LIN {X 0,Y 249.229,Z 243.435,A -85,B 0,C 180,E1 -19068.626,E2 -19068.626} C_VEL
LIN {X 0,Y 249.43,Z 243.409,A -85,B 0,C 180,E1 -19071.911,E2 -19071.911} C_VEL
LIN {X 0,Y 249.274,Z 243.427,A -85,B 0,C 180,E1 -19075.157,E2 -19075.157} C_VEL
LIN {X 0,Y 249.658,Z 243.377,A -85,B 0,C 180,E1 -19078.648,E2 -19078.648} C_VEL
LIN {X 0,Y 249.31,Z 243.427,A -85,B 0,C 180,E1 -19079.548,E2 -19079.548} C_VEL
LIN {X 0,Y 247.865,Z 243.609,A -85,B 0,C 180,E1 -19080.873,E2 -19080.873} C_VEL
LIN {X 0,Y 243.339,Z 244.172,A -85,B 0,C 180,E1 -19083.962,E2 -19083.962} C_VEL
LIN {X 0,Y 242.329,Z 244.29,A -85,B 0,C 180,E1 -19085.35,E2 -19085.35} C_VEL
LIN {X 0,Y 242.288,Z 244.292,A -85,B 0,C 180,E1 -19085.821,E2 -19085.821} C_VEL
LIN {X 0,Y 242.33,Z 244.288,A -85,B 0,C 180,E1 -19089.588,E2 -19089.588} C_VEL
LIN {X 0,Y 242.123,Z 244.317,A -85,B 0,C 180,E1 -19095.152,E2 -19095.152} C_VEL
LIN {X 0,Y 242.026,Z 244.326,A -85,B 0,C 180,E1 -19098.637,E2 -19098.637} C_VEL
LIN {X 0,Y 241.979,Z 244.332,A -85,B 0,C 180,E1 -19102.192,E2 -19102.192} C_VEL
LIN {X 0,Y 241.995,Z 244.332,A -85,B 0,C 180,E1 -19105.834,E2 -19105.834} C_VEL
LIN {X 0,Y 241.972,Z 244.336,A -85,B 0,C 180,E1 -19109.597,E2 -19109.597} C_VEL
LIN {X 0,Y 241.979,Z 244.335,A -85,B 0,C 180,E1 -19113.502,E2 -19113.502} C_VEL
LIN {X 0,Y 241.978,Z 244.34,A -85,B 0,C 180,E1 -19117.593,E2 -19117.593} C_VEL
LIN {X 0,Y 241.892,Z 244.354,A -85,B 0,C 180,E1 -19121.942,E2 -19121.942} C_VEL
LIN {X 0,Y 241.926,Z 244.377,A -85,B 0,C 180,E1 -19125.083,E2 -19125.083} C_VEL
LIN {X 0,Y 244.497,Z 252.638,A -85,B 0,C 180,E1 -19129.628,E2 -19129.628} C_VEL
LIN {X 0,Y 245.734,Z 256.877,A -85,B 0,C 180,E1 -19131.703,E2 -19131.703} C_VEL
LIN {X 0,Y 248.18,Z 261.171,A -85,B 0,C 180,E1 -19132.469,E2 -19132.469} C_VEL
LIN {X 0,Y 251.912,Z 267.851,A -85,B 0,C 180,E1 -19133.592,E2 -19133.592} C_VEL
LIN {X 0,Y 258.214,Z 280.37,A -85,B 0,C 180,E1 -19135.402,E2 -19135.402} C_VEL
LIN {X 0,Y 262.949,Z 291.618,A -85,B 0,C 180,E1 -19136.722,E2 -19136.722} C_VEL
LIN {X 0,Y 265.386,Z 308.755,A -85,B 0,C 180,E1 -19137.801,E2 -19137.801} C_VEL
LIN {X 0,Y 265.835,Z 312.992,A -85,B 0,C 180,E1 -19138.034,E2 -19138.034} C_VEL
LIN {X 0,Y 263.208,Z 366.769,A -85,B 0,C 180,E1 -19139.626,E2 -19139.626} C_VEL
LIN {X 0,Y 261.857,Z 380.21,A -85,B 0,C 180,E1 -19140.286,E2 -19140.286} C_VEL
LIN {X 0,Y 260.056,Z 392.016,A -85,B 0,C 180,E1 -19141.115,E2 -19141.115} C_VEL
LIN {X 0,Y 257.961,Z 403.306,A -85,B 0,C 180,E1 -19142.19,E2 -19142.19} C_VEL
LIN {X 0,Y 255.717,Z 413.719,A -85,B 0,C 180,E1 -19143.475,E2 -19143.475} C_VEL
LIN {X 0,Y 252.935,Z 424.487,A -85,B 0,C 180,E1 -19145.15,E2 -19145.15} C_VEL
LIN {X 0,Y 250.015,Z 435.103,A -85,B 0,C 180,E1 -19147.263,E2 -19147.263} C_VEL
LIN {X 0,Y 247.678,Z 442.971,A -85,B 0,C 180,E1 -19149.227,E2 -19149.227} C_VEL
LIN {X 0,Y 245.365,Z 450.7,A -85,B 0,C 180,E1 -19151.635,E2 -19151.635} C_VEL
LIN {X 0,Y 243.433,Z 456.957,A -85,B 0,C 180,E1 -19154.082,E2 -19154.082} C_VEL
LIN {X 0,Y 241.818,Z 461.955,A -85,B 0,C 180,E1 -19156.556,E2 -19156.556} C_VEL
LIN {X 0,Y 240.833,Z 465.839,A -85,B 0,C 180,E1 -19159.066,E2 -19159.066} C_VEL
LIN {X 0,Y 240.18,Z 468.71,A -85,B 0,C 180,E1 -19161.587,E2 -19161.587} C_VEL
LIN {X 0,Y 239.825,Z 471.07,A -85,B 0,C 180,E1 -19164.957,E2 -19164.957} C_VEL
LIN {X 0,Y 239.808,Z 471.654,A -85,B 0,C 180,E1 -19166.64,E2 -19166.64} C_VEL
LIN {X 0,Y 239.888,Z 471.802,A -85,B 0,C 180,E1 -19168.321,E2 -19168.321} C_VEL
LIN {X 0,Y 239.955,Z 471.553,A -85,B 0,C 180,E1 -19170,E2 -19170} C_VEL
LIN {X 0,Y 239.918,Z 470.902,A -85,B 0,C 180,E1 -19171.679,E2 -19171.679} C_VEL
LIN {X 0,Y 239.837,Z 469.834,A -85,B 0,C 180,E1 -19173.36,E2 -19173.36} C_VEL
LIN {X 0,Y 239.866,Z 468.298,A -85,B 0,C 180,E1 -19175.043,E2 -19175.043} C_VEL
LIN {X 0,Y 240.061,Z 465.178,A -85,B 0,C 180,E1 -19177.57,E2 -19177.57} C_VEL
LIN {X 0,Y 240.512,Z 460.957,A -85,B 0,C 180,E1 -19180.097,E2 -19180.097} C_VEL
LIN {X 0,Y 241.43,Z 454.492,A -85,B 0,C 180,E1 -19183.038,E2 -19183.038} C_VEL
LIN {X 0,Y 242.788,Z 447.431,A -85,B 0,C 180,E1 -19185.531,E2 -19185.531} C_VEL
LIN {X 0,Y 244.421,Z 438.541,A -85,B 0,C 180,E1 -19188.005,E2 -19188.005} C_VEL
LIN {X 0,Y 246.24,Z 428.427,A -85,B 0,C 180,E1 -19190.246,E2 -19190.246} C_VEL
LIN {X 0,Y 248.041,Z 418.09,A -85,B 0,C 180,E1 -19192.05,E2 -19192.05} C_VEL
LIN {X 0,Y 249.916,Z 406.654,A -85,B 0,C 180,E1 -19193.623,E2 -19193.623} C_VEL
LIN {X 0,Y 251.607,Z 394.804,A -85,B 0,C 180,E1 -19194.88,E2 -19194.88} C_VEL
LIN {X 0,Y 252.985,Z 382.547,A -85,B 0,C 180,E1 -19195.836,E2 -19195.836} C_VEL
LIN {X 0,Y 254.124,Z 368.734,A -85,B 0,C 180,E1 -19196.563,E2 -19196.563} C_VEL
LIN {X 0,Y 256.185,Z 310.245,A -85,B 0,C 180,E1 -19198.329,E2 -19198.329} C_VEL
LIN {X 0,Y 251.646,Z 276.723,A -85,B 0,C 180,E1 -19199.901,E2 -19199.901} C_VEL
LIN {X 0,Y 245.317,Z 259.472,A -85,B 0,C 180,E1 -19201.221,E2 -19201.221} C_VEL
LIN {X 0,Y 243.089,Z 248.916,A -85,B 0,C 180,E1 -19205.325,E2 -19205.325} C_VEL
LIN {X 0,Y 242.019,Z 244.338,A -85,B 0,C 180,E1 -19207.219,E2 -19207.219} C_VEL
LIN {X 0,Y 241.893,Z 244.353,A -85,B 0,C 180,E1 -19211.931,E2 -19211.931} C_VEL
LIN {X 0,Y 241.896,Z 244.354,A -85,B 0,C 180,E1 -19216.579,E2 -19216.579} C_VEL
LIN {X 0,Y 241.988,Z 244.344,A -85,B 0,C 180,E1 -19221.641,E2 -19221.641} C_VEL
LIN {X 0,Y 241.987,Z 244.341,A -85,B 0,C 180,E1 -19224.48,E2 -19224.48} C_VEL
LIN {X 0,Y 241.94,Z 244.345,A -85,B 0,C 180,E1 -19228.466,E2 -19228.466} C_VEL
LIN {X 0,Y 241.96,Z 244.343,A -85,B 0,C 180,E1 -19232.298,E2 -19232.298} C_VEL
LIN {X 0,Y 241.989,Z 244.342,A -85,B 0,C 180,E1 -19236,E2 -19236} C_VEL
LIN {X 0,Y 241.989,Z 244.332,A -85,B 0,C 180,E1 -19239.595,E2 -19239.595} C_VEL
LIN {X 0,Y 242.118,Z 244.307,A -85,B 0,C 180,E1 -19243.31,E2 -19243.31} C_VEL
LIN {X 0,Y 242.161,Z 244.319,A -85,B 0,C 180,E1 -19248.27,E2 -19248.27} C_VEL
LIN {X 0,Y 242.356,Z 244.29,A -85,B 0,C 180,E1 -19251.654,E2 -19251.654} C_VEL
LIN {X 0,Y 242.386,Z 244.28,A -85,B 0,C 180,E1 -19253.331,E2 -19253.331} C_VEL
LIN {X 0,Y 242.601,Z 244.245,A -85,B 0,C 180,E1 -19258.331,E2 -19258.331} C_VEL
LIN {X 0,Y 242.609,Z 244.26,A -85,B 0,C 180,E1 -19261.651,E2 -19261.651} C_VEL
LIN {X 0,Y 242.383,Z 244.29,A -85,B 0,C 180,E1 -19266.65,E2 -19266.65} C_VEL
LIN {X 0,Y 242.253,Z 244.302,A -85,B 0,C 180,E1 -19270.014,E2 -19270.014} C_VEL
LIN {X 0,Y 242.121,Z 244.325,A -85,B 0,C 180,E1 -19275.133,E2 -19275.133} C_VEL
LIN {X 0,Y 242.04,Z 244.325,A -85,B 0,C 180,E1 -19278.616,E2 -19278.616} C_VEL
LIN {X 0,Y 241.984,Z 244.339,A -85,B 0,C 180,E1 -19282.171,E2 -19282.171} C_VEL
LIN {X 0,Y 242.025,Z 244.331,A -85,B 0,C 180,E1 -19285.82,E2 -19285.82} C_VEL
LIN {X 0,Y 241.947,Z 244.323,A -85,B 0,C 180,E1 -19289.579,E2 -19289.579} C_VEL
LIN {X 0,Y 241.948,Z 244.325,A -85,B 0,C 180,E1 -19293.484,E2 -19293.484} C_VEL
LIN {X 0,Y 241.95,Z 244.346,A -85,B 0,C 180,E1 -19297.574,E2 -19297.574} C_VEL
LIN {X 0,Y 241.897,Z 244.349,A -85,B 0,C 180,E1 -19301.915,E2 -19301.915} C_VEL
LIN {X 0,Y 241.896,Z 244.352,A -85,B 0,C 180,E1 -19306.563,E2 -19306.563} C_VEL
LIN {X 0,Y 241.914,Z 244.344,A -85,B 0,C 180,E1 -19310.274,E2 -19310.274} C_VEL
LIN {X 0,Y 241.942,Z 244.347,A -85,B 0,C 180,E1 -19314.483,E2 -19314.483} C_VEL
LIN {X 0,Y 241.928,Z 244.349,A -85,B 0,C 180,E1 -19318.474,E2 -19318.474} C_VEL
LIN {X 0,Y 241.962,Z 244.342,A -85,B 0,C 180,E1 -19322.308,E2 -19322.308} C_VEL
LIN {X 0,Y 242.03,Z 244.338,A -85,B 0,C 180,E1 -19326.014,E2 -19326.014} C_VEL
LIN {X 0,Y 242.033,Z 244.34,A -85,B 0,C 180,E1 -19329.608,E2 -19329.608} C_VEL
LIN {X 0,Y 242.112,Z 244.33,A -85,B 0,C 180,E1 -19333.275,E2 -19333.275} C_VEL
LIN {X 0,Y 242.132,Z 244.324,A -85,B 0,C 180,E1 -19338.277,E2 -19338.277} C_VEL
LIN {X 0,Y 242.374,Z 244.292,A -85,B 0,C 180,E1 -19341.664,E2 -19341.664} C_VEL
LIN {X 0,Y 242.215,Z 244.316,A -85,B 0,C 180,E1 -19345.006,E2 -19345.006} C_VEL
LIN {X 0,Y 242.591,Z 244.267,A -85,B 0,C 180,E1 -19348.34,E2 -19348.34} C_VEL
LIN {X 0,Y 242.586,Z 244.266,A -85,B 0,C 180,E1 -19351.608,E2 -19351.608} C_VEL
LIN {X 0,Y 243.555,Z 247.129,A -85,B 0,C 180,E1 -19351.832,E2 -19351.832} C_VEL
LIN {X 0,Y 252.279,Z 267.97,A -85,B 0,C 180,E1 -19353.517,E2 -19353.517} C_VEL
LIN {X 0,Y 257.026,Z 281.714,A -85,B 0,C 180,E1 -19354.454,E2 -19354.454} C_VEL
LIN {X 0,Y 254.486,Z 350.902,A -85,B 0,C 180,E1 -19356.523,E2 -19356.523} C_VEL
LIN {X 0,Y 253.477,Z 364.221,A -85,B 0,C 180,E1 -19357.225,E2 -19357.225} C_VEL
LIN {X 0,Y 252.336,Z 376.71,A -85,B 0,C 180,E1 -19358.206,E2 -19358.206} C_VEL
LIN {X 0,Y 250.849,Z 388.621,A -85,B 0,C 180,E1 -19359.474,E2 -19359.474} C_VEL
LIN {X 0,Y 249.113,Z 400.327,A -85,B 0,C 180,E1 -19361.088,E2 -19361.088} C_VEL
LIN {X 0,Y 247.294,Z 410.881,A -85,B 0,C 180,E1 -19362.932,E2 -19362.932} C_VEL
LIN {X 0,Y 245.507,Z 420.027,A -85,B 0,C 180,E1 -19364.929,E2 -19364.929} C_VEL
LIN {X 0,Y 243.923,Z 428.643,A -85,B 0,C 180,E1 -19367.275,E2 -19367.275} C_VEL
LIN {X 0,Y 242.477,Z 436.333,A -85,B 0,C 180,E1 -19369.911,E2 -19369.911} C_VEL
LIN {X 0,Y 241.496,Z 441.691,A -85,B 0,C 180,E1 -19372.229,E2 -19372.229} C_VEL
LIN {X 0,Y 240.637,Z 446.89,A -85,B 0,C 180,E1 -19375.155,E2 -19375.155} C_VEL
LIN {X 0,Y 240.121,Z 450.46,A -85,B 0,C 180,E1 -19377.923,E2 -19377.923} C_VEL
LIN {X 0,Y 239.71,Z 452.285,A -85,B 0,C 180,E1 -19379.895,E2 -19379.895} C_VEL
LIN {X 0,Y 239.579,Z 453.5,A -85,B 0,C 180,E1 -19381.871,E2 -19381.871} C_VEL
LIN {X 0,Y 239.59,Z 454.308,A -85,B 0,C 180,E1 -19384.803,E2 -19384.803} C_VEL
LIN {X 0,Y 240.039,Z 453.824,A -85,B 0,C 180,E1 -19387.94,E2 -19387.94} C_VEL
LIN {X 0,Y 240.734,Z 452.276,A -85,B 0,C 180,E1 -19390.638,E2 -19390.638} C_VEL
LIN {X 0,Y 241.725,Z 449.574,A -85,B 0,C 180,E1 -19393.394,E2 -19393.394} C_VEL
LIN {X 0,Y 243.197,Z 445.448,A -85,B 0,C 180,E1 -19396.256,E2 -19396.256} C_VEL
LIN {X 0,Y 244.833,Z 440.722,A -85,B 0,C 180,E1 -19398.699,E2 -19398.699} C_VEL
LIN {X 0,Y 246.897,Z 434.429,A -85,B 0,C 180,E1 -19401.242,E2 -19401.242} C_VEL
LIN {X 0,Y 249.516,Z 426.429,A -85,B 0,C 180,E1 -19403.75,E2 -19403.75} C_VEL
LIN {X 0,Y 252.011,Z 418.028,A -85,B 0,C 180,E1 -19405.837,E2 -19405.837} C_VEL
LIN {X 0,Y 254.554,Z 408.571,A -85,B 0,C 180,E1 -19407.726,E2 -19407.726} C_VEL
LIN {X 0,Y 256.971,Z 398.534,A -85,B 0,C 180,E1 -19409.329,E2 -19409.329} C_VEL
LIN {X 0,Y 259.354,Z 386.633,A -85,B 0,C 180,E1 -19410.818,E2 -19410.818} C_VEL
LIN {X 0,Y 261.389,Z 374.238,A -85,B 0,C 180,E1 -19411.988,E2 -19411.988} C_VEL
LIN {X 0,Y 262.934,Z 361.377,A -85,B 0,C 180,E1 -19412.868,E2 -19412.868} C_VEL
LIN {X 0,Y 264.034,Z 347.279,A -85,B 0,C 180,E1 -19413.476,E2 -19413.476} C_VEL
LIN {X 0,Y 266.847,Z 289.944,A -85,B 0,C 180,E1 -19415.15,E2 -19415.15} C_VEL
LIN {X 0,Y 261.533,Z 277.793,A -85,B 0,C 180,E1 -19416.568,E2 -19416.568} C_VEL
LIN {X 0,Y 255.253,Z 265.81,A -85,B 0,C 180,E1 -19418.282,E2 -19418.282} C_VEL
LIN {X 0,Y 248.063,Z 253.948,A -85,B 0,C 180,E1 -19420.373,E2 -19420.373} C_VEL
LIN {X 0,Y 244.555,Z 248.894,A -85,B 0,C 180,E1 -19421.452,E2 -19421.452} C_VEL
LIN {X 0,Y 242.697,Z 246.476,A -85,B 0,C 180,E1 -19422.037,E2 -19422.037} C_VEL
LIN {X 0,Y 242.208,Z 245.036,A -85,B 0,C 180,E1 -19422.273,E2 -19422.273} C_VEL
LIN {X 0,Y 242.093,Z 244.327,A -85,B 0,C 180,E1 -19422.7,E2 -19422.7} C_VEL
LIN {X 0,Y 242.148,Z 244.324,A -85,B 0,C 180,E1 -19426.585,E2 -19426.585} C_VEL
LIN {X 0,Y 242.378,Z 244.286,A -85,B 0,C 180,E1 -19431.674,E2 -19431.674} C_VEL
LIN {X 0,Y 242.234,Z 244.304,A -85,B 0,C 180,E1 -19435.016,E2 -19435.016} C_VEL
LIN {X 0,Y 242.618,Z 244.254,A -85,B 0,C 180,E1 -19438.643,E2 -19438.643} C_VEL
LIN {X 0,Y 242.615,Z 244.254,A -85,B 0,C 180,E1 -19441.669,E2 -19441.669} C_VEL
LIN {X 0,Y 242.288,Z 244.292,A -85,B 0,C 180,E1 -19445.821,E2 -19445.821} C_VEL
LIN {X 0,Y 241.702,Z 244.374,A -85,B 0,C 180,E1 -19447.208,E2 -19447.208} C_VEL
LIN {X 0,Y 240.104,Z 244.573,A -85,B 0,C 180,E1 -19448.569,E2 -19448.569} C_VEL
LIN {X 0,Y 236.234,Z 245.053,A -85,B 0,C 180,E1 -19451.309,E2 -19451.309} C_VEL
LIN {X 0,Y 235.142,Z 245.192,A -85,B 0,C 180,E1 -19452.743,E2 -19452.743} C_VEL
LIN {X 0,Y 235.058,Z 245.195,A -85,B 0,C 180,E1 -19453.229,E2 -19453.229} C_VEL
LIN {X 0,Y 235.012,Z 245.205,A -85,B 0,C 180,E1 -19457.41,E2 -19457.41} C_VEL
LIN {X 0,Y 234.964,Z 245.207,A -85,B 0,C 180,E1 -19461.996,E2 -19461.996} C_VEL
LIN {X 0,Y 234.914,Z 245.212,A -85,B 0,C 180,E1 -19466.673,E2 -19466.673} C_VEL
LIN {X 0,Y 234.897,Z 245.216,A -85,B 0,C 180,E1 -19470.582,E2 -19470.582} C_VEL
LIN {X 0,Y 234.91,Z 245.22,A -85,B 0,C 180,E1 -19474.651,E2 -19474.651} C_VEL
LIN {X 0,Y 234.927,Z 245.22,A -85,B 0,C 180,E1 -19478.942,E2 -19478.942} C_VEL
LIN {X 0,Y 234.87,Z 245.246,A -85,B 0,C 180,E1 -19483.368,E2 -19483.368} C_VEL
LIN {X 0,Y 237.181,Z 252.68,A -85,B 0,C 180,E1 -19487.809,E2 -19487.809} C_VEL
LIN {X 0,Y 238.401,Z 256.511,A -85,B 0,C 180,E1 -19489.819,E2 -19489.819} C_VEL
LIN {X 0,Y 241.18,Z 261.188,A -85,B 0,C 180,E1 -19490.774,E2 -19490.774} C_VEL
LIN {X 0,Y 245.485,Z 268.562,A -85,B 0,C 180,E1 -19492.18,E2 -19492.18} C_VEL
LIN {X 0,Y 251.778,Z 280.727,A -85,B 0,C 180,E1 -19494.115,E2 -19494.115} C_VEL
LIN {X 0,Y 256.961,Z 292.597,A -85,B 0,C 180,E1 -19495.651,E2 -19495.651} C_VEL
LIN {X 0,Y 257.774,Z 294.794,A -85,B 0,C 180,E1 -19495.893,E2 -19495.893} C_VEL
LIN {X 0,Y 260.076,Z 312.12,A -85,B 0,C 180,E1 -19496.998,E2 -19496.998} C_VEL
LIN {X 0,Y 260.14,Z 316.366,A -85,B 0,C 180,E1 -19497.174,E2 -19497.174} C_VEL
LIN {X 0,Y 257.469,Z 367.039,A -85,B 0,C 180,E1 -19498.714,E2 -19498.714} C_VEL
LIN {X 0,Y 255.975,Z 380.852,A -85,B 0,C 180,E1 -19499.418,E2 -19499.418} C_VEL
LIN {X 0,Y 253.918,Z 393.449,A -85,B 0,C 180,E1 -19500.348,E2 -19500.348} C_VEL
LIN {X 0,Y 251.393,Z 405.87,A -85,B 0,C 180,E1 -19501.625,E2 -19501.625} C_VEL
LIN {X 0,Y 248.783,Z 417.027,A -85,B 0,C 180,E1 -19503.129,E2 -19503.129} C_VEL
LIN {X 0,Y 245.965,Z 427.167,A -85,B 0,C 180,E1 -19504.849,E2 -19504.849} C_VEL
LIN {X 0,Y 242.973,Z 437.148,A -85,B 0,C 180,E1 -19507.016,E2 -19507.016} C_VEL
LIN {X 0,Y 240.25,Z 445.98,A -85,B 0,C 180,E1 -19509.45,E2 -19509.45} C_VEL
LIN {X 0,Y 237.974,Z 453.091,A -85,B 0,C 180,E1 -19511.936,E2 -19511.936} C_VEL
LIN {X 0,Y 235.983,Z 458.809,A -85,B 0,C 180,E1 -19514.453,E2 -19514.453} C_VEL
LIN {X 0,Y 234.503,Z 463.345,A -85,B 0,C 180,E1 -19517.011,E2 -19517.011} C_VEL
LIN {X 0,Y 233.574,Z 466.825,A -85,B 0,C 180,E1 -19519.6,E2 -19519.6} C_VEL
LIN {X 0,Y 232.843,Z 469.921,A -85,B 0,C 180,E1 -19523.066,E2 -19523.066} C_VEL
LIN {X 0,Y 232.714,Z 471.074,A -85,B 0,C 180,E1 -19525.356,E2 -19525.356} C_VEL
LIN {X 0,Y 232.798,Z 471.522,A -85,B 0,C 180,E1 -19528.27,E2 -19528.27} C_VEL
LIN {X 0,Y 232.886,Z 471.246,A -85,B 0,C 180,E1 -19530,E2 -19530} C_VEL
LIN {X 0,Y 232.827,Z 470.566,A -85,B 0,C 180,E1 -19531.73,E2 -19531.73} C_VEL
LIN {X 0,Y 232.784,Z 468.23,A -85,B 0,C 180,E1 -19534.853,E2 -19534.853} C_VEL
LIN {X 0,Y 233.013,Z 464.69,A -85,B 0,C 180,E1 -19537.801,E2 -19537.801} C_VEL
LIN {X 0,Y 233.49,Z 460.401,A -85,B 0,C 180,E1 -19540.404,E2 -19540.404} C_VEL
LIN {X 0,Y 234.463,Z 453.861,A -85,B 0,C 180,E1 -19543.433,E2 -19543.433} C_VEL
LIN {X 0,Y 235.873,Z 446.672,A -85,B 0,C 180,E1 -19545.998,E2 -19545.998} C_VEL
LIN {X 0,Y 237.483,Z 438.386,A -85,B 0,C 180,E1 -19548.358,E2 -19548.358} C_VEL
LIN {X 0,Y 239.355,Z 428.438,A -85,B 0,C 180,E1 -19550.63,E2 -19550.63} C_VEL
LIN {X 0,Y 241.193,Z 418.173,A -85,B 0,C 180,E1 -19552.485,E2 -19552.485} C_VEL
LIN {X 0,Y 243.132,Z 406.814,A -85,B 0,C 180,E1 -19554.097,E2 -19554.097} C_VEL
LIN {X 0,Y 244.87,Z 395.08,A -85,B 0,C 180,E1 -19555.386,E2 -19555.386} C_VEL
LIN {X 0,Y 246.366,Z 382.338,A -85,B 0,C 180,E1 -19556.412,E2 -19556.412} C_VEL
LIN {X 0,Y 247.517,Z 368.578,A -85,B 0,C 180,E1 -19557.158,E2 -19557.158} C_VEL
LIN {X 0,Y 249.654,Z 310.988,A -85,B 0,C 180,E1 -19558.942,E2 -19558.942} C_VEL
LIN {X 0,Y 245.413,Z 278.997,A -85,B 0,C 180,E1 -19560.483,E2 -19560.483} C_VEL
LIN {X 0,Y 238,Z 259.227,A -85,B 0,C 180,E1 -19562.068,E2 -19562.068} C_VEL
LIN {X 0,Y 235.926,Z 249.303,A -85,B 0,C 180,E1 -19566.067,E2 -19566.067} C_VEL
LIN {X 0,Y 234.962,Z 245.217,A -85,B 0,C 180,E1 -19567.819,E2 -19567.819} C_VEL
LIN {X 0,Y 234.843,Z 245.232,A -85,B 0,C 180,E1 -19571.558,E2 -19571.558} C_VEL
LIN {X 0,Y 234.861,Z 245.233,A -85,B 0,C 180,E1 -19575.903,E2 -19575.903} C_VEL
LIN {X 0,Y 234.934,Z 245.22,A -85,B 0,C 180,E1 -19581.072,E2 -19581.072} C_VEL
LIN {X 0,Y 234.911,Z 245.224,A -85,B 0,C 180,E1 -19585.349,E2 -19585.349} C_VEL
LIN {X 0,Y 234.897,Z 245.225,A -85,B 0,C 180,E1 -19589.418,E2 -19589.418} C_VEL
LIN {X 0,Y 234.949,Z 245.217,A -85,B 0,C 180,E1 -19593.814,E2 -19593.814} C_VEL
LIN {X 0,Y 234.942,Z 245.214,A -85,B 0,C 180,E1 -19598.954,E2 -19598.954} C_VEL
LIN {X 0,Y 235.06,Z 245.184,A -85,B 0,C 180,E1 -19603.085,E2 -19603.085} C_VEL
LIN {X 0,Y 235.094,Z 245.201,A -85,B 0,C 180,E1 -19607.912,E2 -19607.912} C_VEL
LIN {X 0,Y 235.295,Z 245.172,A -85,B 0,C 180,E1 -19611.402,E2 -19611.402} C_VEL
LIN {X 0,Y 235.337,Z 245.159,A -85,B 0,C 180,E1 -19613.13,E2 -19613.13} C_VEL
LIN {X 0,Y 235.559,Z 245.121,A -85,B 0,C 180,E1 -19618.281,E2 -19618.281} C_VEL
LIN {X 0,Y 235.568,Z 245.136,A -85,B 0,C 180,E1 -19621.7,E2 -19621.7} C_VEL
LIN {X 0,Y 235.335,Z 245.168,A -85,B 0,C 180,E1 -19626.851,E2 -19626.851} C_VEL
LIN {X 0,Y 235.199,Z 245.18,A -85,B 0,C 180,E1 -19630.318,E2 -19630.318} C_VEL
LIN {X 0,Y 235.068,Z 245.202,A -85,B 0,C 180,E1 -19635.598,E2 -19635.598} C_VEL
LIN {X 0,Y 234.979,Z 245.206,A -85,B 0,C 180,E1 -19639.197,E2 -19639.197} C_VEL
LIN {X 0,Y 234.929,Z 245.219,A -85,B 0,C 180,E1 -19642.874,E2 -19642.874} C_VEL
LIN {X 0,Y 234.931,Z 245.213,A -85,B 0,C 180,E1 -19646.65,E2 -19646.65} C_VEL
LIN {X 0,Y 234.873,Z 245.199,A -85,B 0,C 180,E1 -19650.563,E2 -19650.563} C_VEL
LIN {X 0,Y 234.894,Z 245.209,A -85,B 0,C 180,E1 -19654.63,E2 -19654.63} C_VEL
LIN {X 0,Y 234.878,Z 245.226,A -85,B 0,C 180,E1 -19658.927,E2 -19658.927} C_VEL
LIN {X 0,Y 234.85,Z 245.226,A -85,B 0,C 180,E1 -19663.478,E2 -19663.478} C_VEL
LIN {X 0,Y 234.849,Z 245.229,A -85,B 0,C 180,E1 -19666.507,E2 -19666.507} C_VEL
LIN {X 0,Y 234.876,Z 245.223,A -85,B 0,C 180,E1 -19671.071,E2 -19671.071} C_VEL
LIN {X 0,Y 234.885,Z 245.226,A -85,B 0,C 180,E1 -19675.355,E2 -19675.355} C_VEL
LIN {X 0,Y 234.885,Z 245.23,A -85,B 0,C 180,E1 -19679.426,E2 -19679.426} C_VEL
LIN {X 0,Y 234.947,Z 245.221,A -85,B 0,C 180,E1 -19683.789,E2 -19683.789} C_VEL
LIN {X 0,Y 234.999,Z 245.215,A -85,B 0,C 180,E1 -19688.969,E2 -19688.969} C_VEL
LIN {X 0,Y 235.066,Z 245.205,A -85,B 0,C 180,E1 -19693.04,E2 -19693.04} C_VEL
LIN {X 0,Y 235.064,Z 245.204,A -85,B 0,C 180,E1 -19697.92,E2 -19697.92} C_VEL
LIN {X 0,Y 235.324,Z 245.172,A -85,B 0,C 180,E1 -19701.412,E2 -19701.412} C_VEL
LIN {X 0,Y 235.351,Z 245.165,A -85,B 0,C 180,E1 -19703.14,E2 -19703.14} C_VEL
LIN {X 0,Y 235.551,Z 245.144,A -85,B 0,C 180,E1 -19708.29,E2 -19708.29} C_VEL
LIN {X 0,Y 235.566,Z 245.143,A -85,B 0,C 180,E1 -19710.801,E2 -19710.801} C_VEL
LIN {X 0,Y 236.659,Z 248.134,A -85,B 0,C 180,E1 -19711.049,E2 -19711.049} C_VEL
LIN {X 0,Y 244.391,Z 266.1,A -85,B 0,C 180,E1 -19712.599,E2 -19712.599} C_VEL
LIN {X 0,Y 250.582,Z 283.441,A -85,B 0,C 180,E1 -19713.863,E2 -19713.863} C_VEL
LIN {X 0,Y 247.871,Z 351.487,A -85,B 0,C 180,E1 -19715.945,E2 -19715.945} C_VEL
LIN {X 0,Y 246.857,Z 364.37,A -85,B 0,C 180,E1 -19716.641,E2 -19716.641} C_VEL
LIN {X 0,Y 245.626,Z 377.501,A -85,B 0,C 180,E1 -19717.707,E2 -19717.707} C_VEL
LIN {X 0,Y 243.955,Z 390.157,A -85,B 0,C 180,E1 -19719.116,E2 -19719.116} C_VEL
LIN {X 0,Y 242.261,Z 401.018,A -85,B 0,C 180,E1 -19720.677,E2 -19720.677} C_VEL
LIN {X 0,Y 240.488,Z 410.874,A -85,B 0,C 180,E1 -19722.446,E2 -19722.446} C_VEL
LIN {X 0,Y 238.529,Z 420.706,A -85,B 0,C 180,E1 -19724.66,E2 -19724.66} C_VEL
LIN {X 0,Y 236.756,Z 429.889,A -85,B 0,C 180,E1 -19727.268,E2 -19727.268} C_VEL
LIN {X 0,Y 235.486,Z 436.457,A -85,B 0,C 180,E1 -19729.618,E2 -19729.618} C_VEL
LIN {X 0,Y 234.348,Z 442.397,A -85,B 0,C 180,E1 -19732.293,E2 -19732.293} C_VEL
LIN {X 0,Y 233.481,Z 447.737,A -85,B 0,C 180,E1 -19735.471,E2 -19735.471} C_VEL
LIN {X 0,Y 233.029,Z 450.666,A -85,B 0,C 180,E1 -19737.869,E2 -19737.869} C_VEL
LIN {X 0,Y 232.516,Z 453.203,A -85,B 0,C 180,E1 -19740.919,E2 -19740.919} C_VEL
LIN {X 0,Y 232.459,Z 454.16,A -85,B 0,C 180,E1 -19742.969,E2 -19742.969} C_VEL
LIN {X 0,Y 232.541,Z 454.605,A -85,B 0,C 180,E1 -19745.334,E2 -19745.334} C_VEL
LIN {X 0,Y 233.025,Z 454.036,A -85,B 0,C 180,E1 -19748.377,E2 -19748.377} C_VEL
LIN {X 0,Y 233.864,Z 452.253,A -85,B 0,C 180,E1 -19751.385,E2 -19751.385} C_VEL
LIN {X 0,Y 234.986,Z 449.497,A -85,B 0,C 180,E1 -19754.145,E2 -19754.145} C_VEL
LIN {X 0,Y 236.431,Z 445.601,A -85,B 0,C 180,E1 -19756.884,E2 -19756.884} C_VEL
LIN {X 0,Y 238.36,Z 440.461,A -85,B 0,C 180,E1 -19759.574,E2 -19759.574} C_VEL
LIN {X 0,Y 240.633,Z 434.014,A -85,B 0,C 180,E1 -19762.184,E2 -19762.184} C_VEL
LIN {X 0,Y 243.428,Z 425.799,A -85,B 0,C 180,E1 -19764.745,E2 -19764.745} C_VEL
LIN {X 0,Y 246.242,Z 416.682,A -85,B 0,C 180,E1 -19766.992,E2 -19766.992} C_VEL
LIN {X 0,Y 249.052,Z 406.603,A -85,B 0,C 180,E1 -19768.948,E2 -19768.948} C_VEL
LIN {X 0,Y 251.411,Z 396.809,A -85,B 0,C 180,E1 -19770.465,E2 -19770.465} C_VEL
LIN {X 0,Y 253.85,Z 384.799,A -85,B 0,C 180,E1 -19771.935,E2 -19771.935} C_VEL
LIN {X 0,Y 255.814,Z 373.071,A -85,B 0,C 180,E1 -19773.016,E2 -19773.016} C_VEL
LIN {X 0,Y 257.416,Z 359.361,A -85,B 0,C 180,E1 -19773.919,E2 -19773.919} C_VEL
LIN {X 0,Y 258.443,Z 346.379,A -85,B 0,C 180,E1 -19774.453,E2 -19774.453} C_VEL
LIN {X 0,Y 261.287,Z 292.209,A -85,B 0,C 180,E1 -19776.05,E2 -19776.05} C_VEL
LIN {X 0,Y 256.576,Z 281.435,A -85,B 0,C 180,E1 -19777.365,E2 -19777.365} C_VEL
LIN {X 0,Y 250.555,Z 269.811,A -85,B 0,C 180,E1 -19779.11,E2 -19779.11} C_VEL
LIN {X 0,Y 243.712,Z 258.435,A -85,B 0,C 180,E1 -19781.211,E2 -19781.211} C_VEL
LIN {X 0,Y 240.898,Z 254.379,A -85,B 0,C 180,E1 -19782.118,E2 -19782.118} C_VEL
LIN {X 0,Y 238.744,Z 251.324,A -85,B 0,C 180,E1 -19782.836,E2 -19782.836} C_VEL
LIN {X 0,Y 238.047,Z 250.118,A -85,B 0,C 180,E1 -19783.084,E2 -19783.084} C_VEL
LIN {X 0,Y 235.914,Z 247.754,A -85,B 0,C 180,E1 -19783.807,E2 -19783.807} C_VEL
LIN {X 0,Y 235.145,Z 245.471,A -85,B 0,C 180,E1 -19784.2,E2 -19784.2} C_VEL
LIN {X 0,Y 235.094,Z 245.202,A -85,B 0,C 180,E1 -19784.403,E2 -19784.403} C_VEL
LIN {X 0,Y 235.201,Z 245.189,A -85,B 0,C 180,E1 -19789.682,E2 -19789.682} C_VEL
LIN {X 0,Y 235.351,Z 245.17,A -85,B 0,C 180,E1 -19793.15,E2 -19793.15} C_VEL
LIN {X 0,Y 235.584,Z 245.13,A -85,B 0,C 180,E1 -19798.3,E2 -19798.3} C_VEL
LIN {X 0,Y 235.574,Z 245.13,A -85,B 0,C 180,E1 -19801.719,E2 -19801.719} C_VEL
LIN {X 0,Y 235.356,Z 245.158,A -85,B 0,C 180,E1 -19806.869,E2 -19806.869} C_VEL
LIN {X 0,Y 235.212,Z 245.174,A -85,B 0,C 180,E1 -19810.337,E2 -19810.337} C_VEL
LIN {X 0,Y 235.058,Z 245.195,A -85,B 0,C 180,E1 -19813.229,E2 -19813.229} C_VEL
LIN {X 0,Y 234.384,Z 245.279,A -85,B 0,C 180,E1 -19814.659,E2 -19814.659} C_VEL
LIN {X 0,Y 231.467,Z 245.651,A -85,B 0,C 180,E1 -19816.989,E2 -19816.989} C_VEL
LIN {X 0,Y 228.995,Z 245.955,A -85,B 0,C 180,E1 -19818.89,E2 -19818.89} C_VEL
LIN {X 0,Y 227.955,Z 246.089,A -85,B 0,C 180,E1 -19820.367,E2 -19820.367} C_VEL
LIN {X 0,Y 227.881,Z 246.089,A -85,B 0,C 180,E1 -19820.868,E2 -19820.868} C_VEL
LIN {X 0,Y 227.879,Z 246.091,A -85,B 0,C 180,E1 -19825.59,E2 -19825.59} C_VEL
LIN {X 0,Y 227.876,Z 246.09,A -85,B 0,C 180,E1 -19830.284,E2 -19830.284} C_VEL
LIN {X 0,Y 227.881,Z 246.091,A -85,B 0,C 180,E1 -19833.73,E2 -19833.73} C_VEL
LIN {X 0,Y 227.852,Z 246.103,A -85,B 0,C 180,E1 -19838.1,E2 -19838.1} C_VEL
LIN {X 0,Y 227.837,Z 246.197,A -85,B 0,C 180,E1 -19841.467,E2 -19841.467} C_VEL
LIN {X 0,Y 229.992,Z 252.941,A -85,B 0,C 180,E1 -19845.908,E2 -19845.908} C_VEL
LIN {X 0,Y 230.92,Z 255.935,A -85,B 0,C 180,E1 -19847.641,E2 -19847.641} C_VEL
LIN {X 0,Y 233.653,Z 260.418,A -85,B 0,C 180,E1 -19848.695,E2 -19848.695} C_VEL
LIN {X 0,Y 235.113,Z 262.669,A -85,B 0,C 180,E1 -19849.231,E2 -19849.231} C_VEL
LIN {X 0,Y 239.144,Z 269.456,A -85,B 0,C 180,E1 -19850.652,E2 -19850.652} C_VEL
LIN {X 0,Y 242.465,Z 275.361,A -85,B 0,C 180,E1 -19851.771,E2 -19851.771} C_VEL
LIN {X 0,Y 247.809,Z 286.203,A -85,B 0,C 180,E1 -19853.495,E2 -19853.495} C_VEL
LIN {X 0,Y 252.565,Z 297.481,A -85,B 0,C 180,E1 -19854.986,E2 -19854.986} C_VEL
LIN {X 0,Y 254.611,Z 313.592,A -85,B 0,C 180,E1 -19856.046,E2 -19856.046} C_VEL
LIN {X 0,Y 254.357,Z 322.218,A -85,B 0,C 180,E1 -19856.345,E2 -19856.345} C_VEL
LIN {X 0,Y 251.944,Z 366.239,A -85,B 0,C 180,E1 -19857.706,E2 -19857.706} C_VEL
LIN {X 0,Y 250.368,Z 380.278,A -85,B 0,C 180,E1 -19858.421,E2 -19858.421} C_VEL
LIN {X 0,Y 248.226,Z 392.965,A -85,B 0,C 180,E1 -19859.362,E2 -19859.362} C_VEL
LIN {X 0,Y 245.597,Z 405.401,A -85,B 0,C 180,E1 -19860.657,E2 -19860.657} C_VEL
LIN {X 0,Y 243.196,Z 415.278,A -85,B 0,C 180,E1 -19861.993,E2 -19861.993} C_VEL
LIN {X 0,Y 240.197,Z 425.661,A -85,B 0,C 180,E1 -19863.734,E2 -19863.734} C_VEL
LIN {X 0,Y 237.581,Z 434.188,A -85,B 0,C 180,E1 -19865.536,E2 -19865.536} C_VEL
LIN {X 0,Y 234.925,Z 442.123,A -85,B 0,C 180,E1 -19867.579,E2 -19867.579} C_VEL
LIN {X 0,Y 232.504,Z 449.536,A -85,B 0,C 180,E1 -19869.967,E2 -19869.967} C_VEL
LIN {X 0,Y 230.503,Z 455.268,A -85,B 0,C 180,E1 -19872.249,E2 -19872.249} C_VEL
LIN {X 0,Y 228.541,Z 460.502,A -85,B 0,C 180,E1 -19874.848,E2 -19874.848} C_VEL
LIN {X 0,Y 227.195,Z 464.595,A -85,B 0,C 180,E1 -19877.495,E2 -19877.495} C_VEL
LIN {X 0,Y 226.567,Z 466.729,A -85,B 0,C 180,E1 -19879.274,E2 -19879.274} C_VEL
LIN {X 0,Y 225.791,Z 469.757,A -85,B 0,C 180,E1 -19882.848,E2 -19882.848} C_VEL
LIN {X 0,Y 225.612,Z 470.946,A -85,B 0,C 180,E1 -19885.52,E2 -19885.52} C_VEL
LIN {X 0,Y 225.71,Z 471.243,A -85,B 0,C 180,E1 -19888.216,E2 -19888.216} C_VEL
LIN {X 0,Y 225.818,Z 470.939,A -85,B 0,C 180,E1 -19890,E2 -19890} C_VEL
LIN {X 0,Y 225.737,Z 470.222,A -85,B 0,C 180,E1 -19891.784,E2 -19891.784} C_VEL
LIN {X 0,Y 225.698,Z 468.055,A -85,B 0,C 180,E1 -19894.752,E2 -19894.752} C_VEL
LIN {X 0,Y 225.96,Z 464.194,A -85,B 0,C 180,E1 -19898.046,E2 -19898.046} C_VEL
LIN {X 0,Y 226.479,Z 459.833,A -85,B 0,C 180,E1 -19900.73,E2 -19900.73} C_VEL
LIN {X 0,Y 227.338,Z 454.241,A -85,B 0,C 180,E1 -19903.406,E2 -19903.406} C_VEL
LIN {X 0,Y 228.746,Z 447.247,A -85,B 0,C 180,E1 -19906.052,E2 -19906.052} C_VEL
LIN {X 0,Y 230.412,Z 439.069,A -85,B 0,C 180,E1 -19908.505,E2 -19908.505} C_VEL
LIN {X 0,Y 231.898,Z 431.383,A -85,B 0,C 180,E1 -19910.397,E2 -19910.397} C_VEL
LIN {X 0,Y 233.926,Z 420.656,A -85,B 0,C 180,E1 -19912.523,E2 -19912.523} C_VEL
LIN {X 0,Y 235.842,Z 410.036,A -85,B 0,C 180,E1 -19914.188,E2 -19914.188} C_VEL
LIN {X 0,Y 237.689,Z 398.253,A -85,B 0,C 180,E1 -19915.621,E2 -19915.621} C_VEL
LIN {X 0,Y 239.325,Z 386.114,A -85,B 0,C 180,E1 -19916.722,E2 -19916.722} C_VEL
LIN {X 0,Y 240.578,Z 373.003,A -85,B 0,C 180,E1 -19917.57,E2 -19917.57} C_VEL
LIN {X 0,Y 241.434,Z 358.353,A -85,B 0,C 180,E1 -19918.131,E2 -19918.131} C_VEL
LIN {X 0,Y 243.15,Z 311.534,A -85,B 0,C 180,E1 -19919.586,E2 -19919.586} C_VEL
LIN {X 0,Y 239.049,Z 280.971,A -85,B 0,C 180,E1 -19921.124,E2 -19921.124} C_VEL
LIN {X 0,Y 231.981,Z 262.274,A -85,B 0,C 180,E1 -19922.653,E2 -19922.653} C_VEL
LIN {X 0,Y 230.727,Z 258.892,A -85,B 0,C 180,E1 -19922.991,E2 -19922.991} C_VEL
LIN {X 0,Y 228.705,Z 249.435,A -85,B 0,C 180,E1 -19926.956,E2 -19926.956} C_VEL
LIN {X 0,Y 227.893,Z 246.095,A -85,B 0,C 180,E1 -19928.476,E2 -19928.476} C_VEL
LIN {X 0,Y 227.785,Z 246.112,A -85,B 0,C 180,E1 -19932.747,E2 -19932.747} C_VEL
LIN {X 0,Y 227.814,Z 246.11,A -85,B 0,C 180,E1 -19935.196,E2 -19935.196} C_VEL
LIN {X 0,Y 227.838,Z 246.104,A -85,B 0,C 180,E1 -19940.457,E2 -19940.457} C_VEL
LIN {X 0,Y 227.872,Z 246.1,A -85,B 0,C 180,E1 -19944.117,E2 -19944.117} C_VEL
LIN {X 0,Y 227.852,Z 246.1,A -85,B 0,C 180,E1 -19948.365,E2 -19948.365} C_VEL
LIN {X 0,Y 227.843,Z 246.101,A -85,B 0,C 180,E1 -19952.43,E2 -19952.43} C_VEL
LIN {X 0,Y 227.873,Z 246.099,A -85,B 0,C 180,E1 -19956.353,E2 -19956.353} C_VEL
LIN {X 0,Y 227.894,Z 246.083,A -85,B 0,C 180,E1 -19960.161,E2 -19960.161} C_VEL
LIN {X 0,Y 228.022,Z 246.065,A -85,B 0,C 180,E1 -19963.886,E2 -19963.886} C_VEL
LIN {X 0,Y 228.128,Z 246.069,A -85,B 0,C 180,E1 -19969.338,E2 -19969.338} C_VEL
LIN {X 0,Y 228.29,Z 246.039,A -85,B 0,C 180,E1 -19972.917,E2 -19972.917} C_VEL
LIN {X 0,Y 228.492,Z 245.998,A -85,B 0,C 180,E1 -19978.228,E2 -19978.228} C_VEL
LIN {X 0,Y 228.527,Z 246.013,A -85,B 0,C 180,E1 -19981.752,E2 -19981.752} C_VEL
LIN {X 0,Y 228.288,Z 246.047,A -85,B 0,C 180,E1 -19987.063,E2 -19987.063} C_VEL
LIN {X 0,Y 228.129,Z 246.06,A -85,B 0,C 180,E1 -19990.641,E2 -19990.641} C_VEL
LIN {X 0,Y 228.024,Z 246.077,A -85,B 0,C 180,E1 -19996.093,E2 -19996.093} C_VEL
LIN {X 0,Y 227.912,Z 246.09,A -85,B 0,C 180,E1 -19999.816,E2 -19999.816} C_VEL
LIN {X 0,Y 227.88,Z 246.098,A -85,B 0,C 180,E1 -20003.624,E2 -20003.624} C_VEL
LIN {X 0,Y 227.839,Z 246.09,A -85,B 0,C 180,E1 -20007.548,E2 -20007.548} C_VEL
LIN {X 0,Y 227.828,Z 246.071,A -85,B 0,C 180,E1 -20011.615,E2 -20011.615} C_VEL
LIN {X 0,Y 227.833,Z 246.098,A -85,B 0,C 180,E1 -20015.866,E2 -20015.866} C_VEL
LIN {X 0,Y 227.777,Z 246.11,A -85,B 0,C 180,E1 -20020.371,E2 -20020.371} C_VEL
LIN {X 0,Y 227.796,Z 246.107,A -85,B 0,C 180,E1 -20025.185,E2 -20025.185} C_VEL
LIN {X 0,Y 227.785,Z 246.105,A -85,B 0,C 180,E1 -20029.616,E2 -20029.616} C_VEL
LIN {X 0,Y 227.837,Z 246.104,A -85,B 0,C 180,E1 -20034.121,E2 -20034.121} C_VEL
LIN {X 0,Y 227.824,Z 246.106,A -85,B 0,C 180,E1 -20038.372,E2 -20038.372} C_VEL
LIN {X 0,Y 227.839,Z 246.102,A -85,B 0,C 180,E1 -20042.44,E2 -20042.44} C_VEL
LIN {X 0,Y 227.891,Z 246.1,A -85,B 0,C 180,E1 -20046.365,E2 -20046.365} C_VEL
LIN {X 0,Y 227.919,Z 246.097,A -85,B 0,C 180,E1 -20050.173,E2 -20050.173} C_VEL
LIN {X 0,Y 228.012,Z 246.085,A -85,B 0,C 180,E1 -20053.895,E2 -20053.895} C_VEL
LIN {X 0,Y 228.107,Z 246.07,A -85,B 0,C 180,E1 -20059.347,E2 -20059.347} C_VEL
LIN {X 0,Y 228.302,Z 246.043,A -85,B 0,C 180,E1 -20062.927,E2 -20062.927} C_VEL
LIN {X 0,Y 228.507,Z 246.02,A -85,B 0,C 180,E1 -20069.119,E2 -20069.119} C_VEL
LIN {X 0,Y 228.572,Z 246.01,A -85,B 0,C 180,E1 -20069.945,E2 -20069.945} C_VEL
LIN {X 0,Y 229.658,Z 248.995,A -85,B 0,C 180,E1 -20070.21,E2 -20070.21} C_VEL
LIN {X 0,Y 235.235,Z 261.437,A -85,B 0,C 180,E1 -20071.367,E2 -20071.367} C_VEL
LIN {X 0,Y 240.979,Z 275.922,A -85,B 0,C 180,E1 -20072.56,E2 -20072.56} C_VEL
LIN {X 0,Y 244.054,Z 285.524,A -85,B 0,C 180,E1 -20073.242,E2 -20073.242} C_VEL
LIN {X 0,Y 241.343,Z 351.055,A -85,B 0,C 180,E1 -20075.288,E2 -20075.288} C_VEL
LIN {X 0,Y 240.237,Z 364.913,A -85,B 0,C 180,E1 -20076.054,E2 -20076.054} C_VEL
LIN {X 0,Y 239.03,Z 377.217,A -85,B 0,C 180,E1 -20077.072,E2 -20077.072} C_VEL
LIN {X 0,Y 237.575,Z 388.26,A -85,B 0,C 180,E1 -20078.291,E2 -20078.291} C_VEL
LIN {X 0,Y 235.811,Z 399.378,A -85,B 0,C 180,E1 -20079.867,E2 -20079.867} C_VEL
LIN {X 0,Y 233.947,Z 409.667,A -85,B 0,C 180,E1 -20081.699,E2 -20081.699} C_VEL
LIN {X 0,Y 232.213,Z 418.186,A -85,B 0,C 180,E1 -20083.565,E2 -20083.565} C_VEL
LIN {X 0,Y 230.49,Z 426.921,A -85,B 0,C 180,E1 -20085.927,E2 -20085.927} C_VEL
LIN {X 0,Y 228.945,Z 434.243,A -85,B 0,C 180,E1 -20088.399,E2 -20088.399} C_VEL
LIN {X 0,Y 227.624,Z 440.97,A -85,B 0,C 180,E1 -20091.271,E2 -20091.271} C_VEL
LIN {X 0,Y 226.814,Z 445.529,A -85,B 0,C 180,E1 -20093.753,E2 -20093.753} C_VEL
LIN {X 0,Y 226.199,Z 449.746,A -85,B 0,C 180,E1 -20096.775,E2 -20096.775} C_VEL
LIN {X 0,Y 225.539,Z 452.738,A -85,B 0,C 180,E1 -20099.905,E2 -20099.905} C_VEL
LIN {X 0,Y 225.36,Z 454.288,A -85,B 0,C 180,E1 -20102.671,E2 -20102.671} C_VEL
LIN {X 0,Y 225.508,Z 454.856,A -85,B 0,C 180,E1 -20105.897,E2 -20105.897} C_VEL
LIN {X 0,Y 226.078,Z 454.178,A -85,B 0,C 180,E1 -20109.019,E2 -20109.019} C_VEL
LIN {X 0,Y 226.988,Z 452.365,A -85,B 0,C 180,E1 -20112.024,E2 -20112.024} C_VEL
LIN {X 0,Y 228.321,Z 449.299,A -85,B 0,C 180,E1 -20115.068,E2 -20115.068} C_VEL
LIN {X 0,Y 229.84,Z 445.466,A -85,B 0,C 180,E1 -20117.74,E2 -20117.74} C_VEL
LIN {X 0,Y 231.936,Z 440.212,A -85,B 0,C 180,E1 -20120.497,E2 -20120.497} C_VEL
LIN {X 0,Y 234.46,Z 433.526,A -85,B 0,C 180,E1 -20123.18,E2 -20123.18} C_VEL
LIN {X 0,Y 237.393,Z 425.199,A -85,B 0,C 180,E1 -20125.786,E2 -20125.786} C_VEL
LIN {X 0,Y 240.299,Z 416.214,A -85,B 0,C 180,E1 -20128.01,E2 -20128.01} C_VEL
LIN {X 0,Y 243.348,Z 405.692,A -85,B 0,C 180,E1 -20130.042,E2 -20130.042} C_VEL
LIN {X 0,Y 246.022,Z 394.976,A -85,B 0,C 180,E1 -20131.677,E2 -20131.677} C_VEL
LIN {X 0,Y 248.205,Z 384.593,A -85,B 0,C 180,E1 -20132.928,E2 -20132.928} C_VEL
LIN {X 0,Y 250.191,Z 372.914,A -85,B 0,C 180,E1 -20134.01,E2 -20134.01} C_VEL
LIN {X 0,Y 251.756,Z 360.067,A -85,B 0,C 180,E1 -20134.87,E2 -20134.87} C_VEL
LIN {X 0,Y 252.898,Z 346.326,A -85,B 0,C 180,E1 -20135.445,E2 -20135.445} C_VEL
LIN {X 0,Y 255.752,Z 294.415,A -85,B 0,C 180,E1 -20136.998,E2 -20136.998} C_VEL
LIN {X 0,Y 251.203,Z 284.035,A -85,B 0,C 180,E1 -20138.359,E2 -20138.359} C_VEL
LIN {X 0,Y 245.542,Z 273.121,A -85,B 0,C 180,E1 -20140.088,E2 -20140.088} C_VEL
LIN {X 0,Y 239.719,Z 263.372,A -85,B 0,C 180,E1 -20141.986,E2 -20141.986} C_VEL
LIN {X 0,Y 237.02,Z 259.535,A -85,B 0,C 180,E1 -20142.89,E2 -20142.89} C_VEL
LIN {X 0,Y 234.22,Z 255.477,A -85,B 0,C 180,E1 -20143.889,E2 -20143.889} C_VEL
LIN {X 0,Y 232.031,Z 252.443,A -85,B 0,C 180,E1 -20144.699,E2 -20144.699} C_VEL
LIN {X 0,Y 231.169,Z 251.116,A -85,B 0,C 180,E1 -20145.035,E2 -20145.035} C_VEL
LIN {X 0,Y 228.979,Z 248.843,A -85,B 0,C 180,E1 -20145.854,E2 -20145.854} C_VEL
LIN {X 0,Y 228.041,Z 246.079,A -85,B 0,C 180,E1 -20146.363,E2 -20146.363} C_VEL
LIN {X 0,Y 228.248,Z 246.046,A -85,B 0,C 180,E1 -20151.154,E2 -20151.154} C_VEL
LIN {X 0,Y 228.302,Z 246.047,A -85,B 0,C 180,E1 -20152.937,E2 -20152.937} C_VEL
LIN {X 0,Y 228.543,Z 246.007,A -85,B 0,C 180,E1 -20158.248,E2 -20158.248} C_VEL
LIN {X 0,Y 228.532,Z 246.007,A -85,B 0,C 180,E1 -20161.772,E2 -20161.772} C_VEL
LIN {X 0,Y 228.309,Z 246.038,A -85,B 0,C 180,E1 -20167.083,E2 -20167.083} C_VEL
LIN {X 0,Y 228.143,Z 246.055,A -85,B 0,C 180,E1 -20170.661,E2 -20170.661} C_VEL
LIN {X 0,Y 228.021,Z 246.082,A -85,B 0,C 180,E1 -20176.114,E2 -20176.114} C_VEL
LIN {X 0,Y 227.881,Z 246.089,A -85,B 0,C 180,E1 -20180.868,E2 -20180.868} C_VEL
LIN {X 0,Y 227.248,Z 246.17,A -85,B 0,C 180,E1 -20182.343,E2 -20182.343} C_VEL
LIN {X 0,Y 224.421,Z 246.534,A -85,B 0,C 180,E1 -20184.749,E2 -20184.749} C_VEL
LIN {X 0,Y 221.141,Z 246.944,A -85,B 0,C 180,E1 -20187.721,E2 -20187.721} C_VEL
LIN {X 0,Y 220.788,Z 246.979,A -85,B 0,C 180,E1 -20188.752,E2 -20188.752} C_VEL
LIN {X 0,Y 220.814,Z 246.974,A -85,B 0,C 180,E1 -20192.767,E2 -20192.767} C_VEL
LIN {X 0,Y 220.81,Z 246.974,A -85,B 0,C 180,E1 -20197.28,E2 -20197.28} C_VEL
LIN {X 0,Y 220.801,Z 247.092,A -85,B 0,C 180,E1 -20199.253,E2 -20199.253} C_VEL
LIN {X 0,Y 222.879,Z 253.489,A -85,B 0,C 180,E1 -20203.936,E2 -20203.936} C_VEL
LIN {X 0,Y 223.597,Z 255.581,A -85,B 0,C 180,E1 -20205.207,E2 -20205.207} C_VEL
LIN {X 0,Y 226.469,Z 260.172,A -85,B 0,C 180,E1 -20206.463,E2 -20206.463} C_VEL
LIN {X 0,Y 228.091,Z 262.613,A -85,B 0,C 180,E1 -20207.129,E2 -20207.129} C_VEL
LIN {X 0,Y 231.532,Z 268.019,A -85,B 0,C 180,E1 -20208.479,E2 -20208.479} C_VEL
LIN {X 0,Y 236.855,Z 277.156,A -85,B 0,C 180,E1 -20210.432,E2 -20210.432} C_VEL
LIN {X 0,Y 242.925,Z 289.493,A -85,B 0,C 180,E1 -20212.538,E2 -20212.538} C_VEL
LIN {X 0,Y 247.568,Z 300.712,A -85,B 0,C 180,E1 -20214.075,E2 -20214.075} C_VEL
LIN {X 0,Y 249.276,Z 315.512,A -85,B 0,C 180,E1 -20215.072,E2 -20215.072} C_VEL
LIN {X 0,Y 246.331,Z 367.032,A -85,B 0,C 180,E1 -20216.718,E2 -20216.718} C_VEL
LIN {X 0,Y 244.747,Z 380.428,A -85,B 0,C 180,E1 -20217.425,E2 -20217.425} C_VEL
LIN {X 0,Y 242.596,Z 392.481,A -85,B 0,C 180,E1 -20218.327,E2 -20218.327} C_VEL
LIN {X 0,Y 239.866,Z 404.966,A -85,B 0,C 180,E1 -20219.642,E2 -20219.642} C_VEL
LIN {X 0,Y 237.282,Z 414.883,A -85,B 0,C 180,E1 -20220.988,E2 -20220.988} C_VEL
LIN {X 0,Y 234.199,Z 425.283,A -85,B 0,C 180,E1 -20222.766,E2 -20222.766} C_VEL
LIN {X 0,Y 231.161,Z 434.708,A -85,B 0,C 180,E1 -20224.809,E2 -20224.809} C_VEL
LIN {X 0,Y 227.911,Z 443.839,A -85,B 0,C 180,E1 -20227.329,E2 -20227.329} C_VEL
LIN {X 0,Y 225.254,Z 451.235,A -85,B 0,C 180,E1 -20229.929,E2 -20229.929} C_VEL
LIN {X 0,Y 223.01,Z 457.22,A -85,B 0,C 180,E1 -20232.58,E2 -20232.58} C_VEL
LIN {X 0,Y 221.086,Z 461.985,A -85,B 0,C 180,E1 -20235.268,E2 -20235.268} C_VEL
LIN {X 0,Y 219.861,Z 465.652,A -85,B 0,C 180,E1 -20238.008,E2 -20238.008} C_VEL
LIN {X 0,Y 219.044,Z 468.324,A -85,B 0,C 180,E1 -20240.769,E2 -20240.769} C_VEL
LIN {X 0,Y 218.713,Z 469.606,A -85,B 0,C 180,E1 -20242.615,E2 -20242.615} C_VEL
LIN {X 0,Y 218.539,Z 470.795,A -85,B 0,C 180,E1 -20245.598,E2 -20245.598} C_VEL
LIN {X 0,Y 218.623,Z 470.963,A -85,B 0,C 180,E1 -20248.158,E2 -20248.158} C_VEL
LIN {X 0,Y 218.729,Z 470.629,A -85,B 0,C 180,E1 -20250,E2 -20250} C_VEL
LIN {X 0,Y 218.65,Z 469.86,A -85,B 0,C 180,E1 -20251.842,E2 -20251.842} C_VEL
LIN {X 0,Y 218.602,Z 467.909,A -85,B 0,C 180,E1 -20254.609,E2 -20254.609} C_VEL
LIN {X 0,Y 218.799,Z 464.946,A -85,B 0,C 180,E1 -20257.382,E2 -20257.382} C_VEL
LIN {X 0,Y 219.237,Z 460.896,A -85,B 0,C 180,E1 -20260.155,E2 -20260.155} C_VEL
LIN {X 0,Y 220.196,Z 454.619,A -85,B 0,C 180,E1 -20263.379,E2 -20263.379} C_VEL
LIN {X 0,Y 221.637,Z 447.77,A -85,B 0,C 180,E1 -20266.108,E2 -20266.108} C_VEL
LIN {X 0,Y 223.444,Z 439.107,A -85,B 0,C 180,E1 -20268.838,E2 -20268.838} C_VEL
LIN {X 0,Y 225.218,Z 430.375,A -85,B 0,C 180,E1 -20271.03,E2 -20271.03} C_VEL
LIN {X 0,Y 227.304,Z 419.49,A -85,B 0,C 180,E1 -20273.217,E2 -20273.217} C_VEL
LIN {X 0,Y 229.321,Z 408.631,A -85,B 0,C 180,E1 -20274.922,E2 -20274.922} C_VEL
LIN {X 0,Y 231.295,Z 396.492,A -85,B 0,C 180,E1 -20276.384,E2 -20276.384} C_VEL
LIN {X 0,Y 232.78,Z 385.174,A -85,B 0,C 180,E1 -20277.414,E2 -20277.414} C_VEL
LIN {X 0,Y 234.028,Z 372.705,A -85,B 0,C 180,E1 -20278.227,E2 -20278.227} C_VEL
LIN {X 0,Y 234.9,Z 358.671,A -85,B 0,C 180,E1 -20278.78,E2 -20278.78} C_VEL
LIN {X 0,Y 236.695,Z 312.67,A -85,B 0,C 180,E1 -20280.244,E2 -20280.244} C_VEL
LIN {X 0,Y 232.755,Z 283.043,A -85,B 0,C 180,E1 -20281.78,E2 -20281.78} C_VEL
LIN {X 0,Y 226.031,Z 265.249,A -85,B 0,C 180,E1 -20283.289,E2 -20283.289} C_VEL
LIN {X 0,Y 223.467,Z 258.65,A -85,B 0,C 180,E1 -20283.93,E2 -20283.93} C_VEL
LIN {X 0,Y 221.64,Z 250.376,A -85,B 0,C 180,E1 -20287.547,E2 -20287.547} C_VEL
LIN {X 0,Y 220.819,Z 246.976,A -85,B 0,C 180,E1 -20289.128,E2 -20289.128} C_VEL
LIN {X 0,Y 220.758,Z 246.99,A -85,B 0,C 180,E1 -20294.457,E2 -20294.457} C_VEL
LIN {X 0,Y 220.747,Z 246.988,A -85,B 0,C 180,E1 -20298.031,E2 -20298.031} C_VEL
LIN {X 0,Y 220.841,Z 246.976,A -85,B 0,C 180,E1 -20302.786,E2 -20302.786} C_VEL
LIN {X 0,Y 220.815,Z 246.981,A -85,B 0,C 180,E1 -20307.234,E2 -20307.234} C_VEL
LIN {X 0,Y 220.802,Z 246.983,A -85,B 0,C 180,E1 -20311.472,E2 -20311.472} C_VEL
LIN {X 0,Y 220.811,Z 246.98,A -85,B 0,C 180,E1 -20315.549,E2 -20315.549} C_VEL
LIN {X 0,Y 220.853,Z 246.963,A -85,B 0,C 180,E1 -20319.5,E2 -20319.5} C_VEL
LIN {X 0,Y 220.98,Z 246.936,A -85,B 0,C 180,E1 -20323.358,E2 -20323.358} C_VEL
LIN {X 0,Y 221.054,Z 246.948,A -85,B 0,C 180,E1 -20328.993,E2 -20328.993} C_VEL
LIN {X 0,Y 221.227,Z 246.918,A -85,B 0,C 180,E1 -20332.69,E2 -20332.69} C_VEL
LIN {X 0,Y 221.429,Z 246.874,A -85,B 0,C 180,E1 -20338.171,E2 -20338.171} C_VEL
LIN {X 0,Y 221.533,Z 246.875,A -85,B 0,C 180,E1 -20339.99,E2 -20339.99} C_VEL
LIN {X 0,Y 221.46,Z 246.894,A -85,B 0,C 180,E1 -20341.808,E2 -20341.808} C_VEL
LIN {X 0,Y 221.226,Z 246.926,A -85,B 0,C 180,E1 -20347.29,E2 -20347.29} C_VEL
LIN {X 0,Y 221.049,Z 246.943,A -85,B 0,C 180,E1 -20350.986,E2 -20350.986} C_VEL
LIN {X 0,Y 220.99,Z 246.952,A -85,B 0,C 180,E1 -20356.62,E2 -20356.62} C_VEL
LIN {X 0,Y 220.861,Z 246.967,A -85,B 0,C 180,E1 -20360.477,E2 -20360.477} C_VEL
LIN {X 0,Y 220.833,Z 246.973,A -85,B 0,C 180,E1 -20364.426,E2 -20364.426} C_VEL
LIN {X 0,Y 220.784,Z 246.965,A -85,B 0,C 180,E1 -20368.507,E2 -20368.507} C_VEL
LIN {X 0,Y 220.783,Z 246.951,A -85,B 0,C 180,E1 -20372.747,E2 -20372.747} C_VEL
LIN {X 0,Y 220.769,Z 246.98,A -85,B 0,C 180,E1 -20377.266,E2 -20377.266} C_VEL
LIN {X 0,Y 220.729,Z 246.985,A -85,B 0,C 180,E1 -20381.945,E2 -20381.945} C_VEL
LIN {X 0,Y 220.736,Z 246.989,A -85,B 0,C 180,E1 -20385.538,E2 -20385.538} C_VEL
LIN {X 0,Y 220.766,Z 246.978,A -85,B 0,C 180,E1 -20390.455,E2 -20390.455} C_VEL
LIN {X 0,Y 220.758,Z 246.988,A -85,B 0,C 180,E1 -20395.038,E2 -20395.038} C_VEL
LIN {X 0,Y 220.824,Z 246.982,A -85,B 0,C 180,E1 -20399.389,E2 -20399.389} C_VEL
LIN {X 0,Y 220.849,Z 246.978,A -85,B 0,C 180,E1 -20403.544,E2 -20403.544} C_VEL
LIN {X 0,Y 220.894,Z 246.97,A -85,B 0,C 180,E1 -20407.556,E2 -20407.556} C_VEL
LIN {X 0,Y 220.943,Z 246.962,A -85,B 0,C 180,E1 -20412.561,E2 -20412.561} C_VEL
LIN {X 0,Y 220.959,Z 246.962,A -85,B 0,C 180,E1 -20417.136,E2 -20417.136} C_VEL
LIN {X 0,Y 221.184,Z 246.934,A -85,B 0,C 180,E1 -20420.859,E2 -20420.859} C_VEL
LIN {X 0,Y 221.237,Z 246.923,A -85,B 0,C 180,E1 -20422.7,E2 -20422.7} C_VEL
LIN {X 0,Y 221.485,Z 246.973,A -85,B 0,C 180,E1 -20429.033,E2 -20429.033} C_VEL
LIN {X 0,Y 222.502,Z 249.754,A -85,B 0,C 180,E1 -20429.286,E2 -20429.286} C_VEL
LIN {X 0,Y 228.073,Z 261.418,A -85,B 0,C 180,E1 -20430.481,E2 -20430.481} C_VEL
LIN {X 0,Y 234.747,Z 278.139,A -85,B 0,C 180,E1 -20431.924,E2 -20431.924} C_VEL
LIN {X 0,Y 237.564,Z 286.455,A -85,B 0,C 180,E1 -20432.549,E2 -20432.549} C_VEL
LIN {X 0,Y 234.729,Z 352.153,A -85,B 0,C 180,E1 -20434.668,E2 -20434.668} C_VEL
LIN {X 0,Y 233.688,Z 364.812,A -85,B 0,C 180,E1 -20435.39,E2 -20435.39} C_VEL
LIN {X 0,Y 232.387,Z 377.755,A -85,B 0,C 180,E1 -20436.489,E2 -20436.489} C_VEL
LIN {X 0,Y 230.695,Z 389.785,A -85,B 0,C 180,E1 -20437.879,E2 -20437.879} C_VEL
LIN {X 0,Y 228.82,Z 401,A -85,B 0,C 180,E1 -20439.552,E2 -20439.552} C_VEL
LIN {X 0,Y 226.978,Z 410.789,A -85,B 0,C 180,E1 -20441.384,E2 -20441.384} C_VEL
LIN {X 0,Y 225.025,Z 419.876,A -85,B 0,C 180,E1 -20443.486,E2 -20443.486} C_VEL
LIN {X 0,Y 223.257,Z 428.5,A -85,B 0,C 180,E1 -20445.988,E2 -20445.988} C_VEL
LIN {X 0,Y 221.749,Z 435.432,A -85,B 0,C 180,E1 -20448.477,E2 -20448.477} C_VEL
LIN {X 0,Y 220.476,Z 441.818,A -85,B 0,C 180,E1 -20451.36,E2 -20451.36} C_VEL
LIN {X 0,Y 219.473,Z 447.256,A -85,B 0,C 180,E1 -20454.6,E2 -20454.6} C_VEL
LIN {X 0,Y 218.843,Z 451.066,A -85,B 0,C 180,E1 -20457.752,E2 -20457.752} C_VEL
LIN {X 0,Y 218.326,Z 453.651,A -85,B 0,C 180,E1 -20460.999,E2 -20460.999} C_VEL
LIN {X 0,Y 218.247,Z 454.66,A -85,B 0,C 180,E1 -20463.19,E2 -20463.19} C_VEL
LIN {X 0,Y 218.507,Z 455.106,A -85,B 0,C 180,E1 -20466.499,E2 -20466.499} C_VEL
LIN {X 0,Y 219.212,Z 454.252,A -85,B 0,C 180,E1 -20469.88,E2 -20469.88} C_VEL
LIN {X 0,Y 220.189,Z 452.416,A -85,B 0,C 180,E1 -20472.786,E2 -20472.786} C_VEL
LIN {X 0,Y 221.55,Z 449.43,A -85,B 0,C 180,E1 -20475.76,E2 -20475.76} C_VEL
LIN {X 0,Y 223.554,Z 444.746,A -85,B 0,C 180,E1 -20478.98,E2 -20478.98} C_VEL
LIN {X 0,Y 225.884,Z 439.083,A -85,B 0,C 180,E1 -20481.856,E2 -20481.856} C_VEL
LIN {X 0,Y 228.297,Z 433.13,A -85,B 0,C 180,E1 -20484.219,E2 -20484.219} C_VEL
LIN {X 0,Y 231.485,Z 424.634,A -85,B 0,C 180,E1 -20486.888,E2 -20486.888} C_VEL
LIN {X 0,Y 234.456,Z 415.845,A -85,B 0,C 180,E1 -20489.052,E2 -20489.052} C_VEL
LIN {X 0,Y 237.284,Z 406.49,A -85,B 0,C 180,E1 -20490.894,E2 -20490.894} C_VEL
LIN {X 0,Y 240.106,Z 395.749,A -85,B 0,C 180,E1 -20492.578,E2 -20492.578} C_VEL
LIN {X 0,Y 242.529,Z 384.734,A -85,B 0,C 180,E1 -20493.935,E2 -20493.935} C_VEL
LIN {X 0,Y 244.615,Z 372.902,A -85,B 0,C 180,E1 -20495.039,E2 -20495.039} C_VEL
LIN {X 0,Y 246.315,Z 359.683,A -85,B 0,C 180,E1 -20495.925,E2 -20495.925} C_VEL
LIN {X 0,Y 247.455,Z 346.056,A -85,B 0,C 180,E1 -20496.494,E2 -20496.494} C_VEL
LIN {X 0,Y 250.281,Z 296.486,A -85,B 0,C 180,E1 -20498.02,E2 -20498.02} C_VEL
LIN {X 0,Y 245.259,Z 285.359,A -85,B 0,C 180,E1 -20499.601,E2 -20499.601} C_VEL
LIN {X 0,Y 240.59,Z 276.405,A -85,B 0,C 180,E1 -20501.135,E2 -20501.135} C_VEL
LIN {X 0,Y 235.612,Z 268.082,A -85,B 0,C 180,E1 -20502.842,E2 -20502.842} C_VEL
LIN {X 0,Y 233.044,Z 264.39,A -85,B 0,C 180,E1 -20503.759,E2 -20503.759} C_VEL
LIN {X 0,Y 230.648,Z 260.865,A -85,B 0,C 180,E1 -20504.661,E2 -20504.661} C_VEL
LIN {X 0,Y 227.792,Z 256.877,A -85,B 0,C 180,E1 -20505.779,E2 -20505.779} C_VEL
LIN {X 0,Y 225.481,Z 253.955,A -85,B 0,C 180,E1 -20506.722,E2 -20506.722} C_VEL
LIN {X 0,Y 224.592,Z 252.284,A -85,B 0,C 180,E1 -20507.128,E2 -20507.128} C_VEL
LIN {X 0,Y 222.274,Z 250.158,A -85,B 0,C 180,E1 -20508.095,E2 -20508.095} C_VEL
LIN {X 0,Y 221.249,Z 248.011,A -85,B 0,C 180,E1 -20508.619,E2 -20508.619} C_VEL
LIN {X 0,Y 221.04,Z 246.946,A -85,B 0,C 180,E1 -20508.782,E2 -20508.782} C_VEL
LIN {X 0,Y 221.239,Z 246.925,A -85,B 0,C 180,E1 -20512.711,E2 -20512.711} C_VEL
LIN {X 0,Y 221.501,Z 246.884,A -85,B 0,C 180,E1 -20518.192,E2 -20518.192} C_VEL
LIN {X 0,Y 221.465,Z 246.887,A -85,B 0,C 180,E1 -20521.829,E2 -20521.829} C_VEL
LIN {X 0,Y 221.246,Z 246.919,A -85,B 0,C 180,E1 -20527.31,E2 -20527.31} C_VEL
LIN {X 0,Y 221.063,Z 246.939,A -85,B 0,C 180,E1 -20531.006,E2 -20531.006} C_VEL
LIN {X 0,Y 220.98,Z 246.959,A -85,B 0,C 180,E1 -20536.642,E2 -20536.642} C_VEL
LIN {X 0,Y 220.836,Z 246.973,A -85,B 0,C 180,E1 -20540.851,E2 -20540.851} C_VEL
LIN {X 0,Y 220.81,Z 246.979,A -85,B 0,C 180,E1 -20544.451,E2 -20544.451} C_VEL
LIN {X 0,Y 220.788,Z 246.979,A -85,B 0,C 180,E1 -20548.752,E2 -20548.752} C_VEL
LIN {X 0,Y 220.084,Z 247.062,A -85,B 0,C 180,E1 -20549.765,E2 -20549.765} C_VEL
LIN {X 0,Y 217.254,Z 247.419,A -85,B 0,C 180,E1 -20551.359,E2 -20551.359} C_VEL
LIN {X 0,Y 214.425,Z 247.769,A -85,B 0,C 180,E1 -20552.993,E2 -20552.993} C_VEL
LIN {X 0,Y 213.76,Z 247.85,A -85,B 0,C 180,E1 -20554.052,E2 -20554.052} C_VEL
LIN {X 0,Y 213.78,Z 247.949,A -85,B 0,C 180,E1 -20556.636,E2 -20556.636} C_VEL
LIN {X 0,Y 215.645,Z 253.747,A -85,B 0,C 180,E1 -20561.447,E2 -20561.447} C_VEL
LIN {X 0,Y 216.118,Z 255.098,A -85,B 0,C 180,E1 -20562.289,E2 -20562.289} C_VEL
LIN {X 0,Y 219.861,Z 260.508,A -85,B 0,C 180,E1 -20564.145,E2 -20564.145} C_VEL
LIN {X 0,Y 224.861,Z 268.273,A -85,B 0,C 180,E1 -20566.401,E2 -20566.401} C_VEL
LIN {X 0,Y 228.173,Z 273.681,A -85,B 0,C 180,E1 -20567.771,E2 -20567.771} C_VEL
LIN {X 0,Y 233.241,Z 282.703,A -85,B 0,C 180,E1 -20569.739,E2 -20569.739} C_VEL
LIN {X 0,Y 238.695,Z 294.133,A -85,B 0,C 180,E1 -20571.729,E2 -20571.729} C_VEL
LIN {X 0,Y 242.538,Z 303.592,A -85,B 0,C 180,E1 -20573.088,E2 -20573.088} C_VEL
LIN {X 0,Y 244.014,Z 317.147,A -85,B 0,C 180,E1 -20574.023,E2 -20574.023} C_VEL
LIN {X 0,Y 241.016,Z 366.309,A -85,B 0,C 180,E1 -20575.605,E2 -20575.605} C_VEL
LIN {X 0,Y 239.303,Z 380.109,A -85,B 0,C 180,E1 -20576.336,E2 -20576.336} C_VEL
LIN {X 0,Y 237.069,Z 392.133,A -85,B 0,C 180,E1 -20577.248,E2 -20577.248} C_VEL
LIN {X 0,Y 234.235,Z 404.592,A -85,B 0,C 180,E1 -20578.58,E2 -20578.58} C_VEL
LIN {X 0,Y 231.151,Z 415.772,A -85,B 0,C 180,E1 -20580.142,E2 -20580.142} C_VEL
LIN {X 0,Y 227.949,Z 425.962,A -85,B 0,C 180,E1 -20581.955,E2 -20581.955} C_VEL
LIN {X 0,Y 224.787,Z 435.177,A -85,B 0,C 180,E1 -20584.043,E2 -20584.043} C_VEL
LIN {X 0,Y 221.384,Z 444.183,A -85,B 0,C 180,E1 -20586.621,E2 -20586.621} C_VEL
LIN {X 0,Y 218.61,Z 451.474,A -85,B 0,C 180,E1 -20589.291,E2 -20589.291} C_VEL
LIN {X 0,Y 216.244,Z 457.353,A -85,B 0,C 180,E1 -20592.016,E2 -20592.016} C_VEL
LIN {X 0,Y 214.217,Z 462.02,A -85,B 0,C 180,E1 -20594.784,E2 -20594.784} C_VEL
LIN {X 0,Y 212.89,Z 465.603,A -85,B 0,C 180,E1 -20597.61,E2 -20597.61} C_VEL
LIN {X 0,Y 212.028,Z 468.207,A -85,B 0,C 180,E1 -20600.461,E2 -20600.461} C_VEL
LIN {X 0,Y 211.654,Z 469.443,A -85,B 0,C 180,E1 -20602.368,E2 -20602.368} C_VEL
LIN {X 0,Y 211.446,Z 470.606,A -85,B 0,C 180,E1 -20605.76,E2 -20605.76} C_VEL
LIN {X 0,Y 211.519,Z 470.681,A -85,B 0,C 180,E1 -20608.096,E2 -20608.096} C_VEL
LIN {X 0,Y 211.642,Z 470.31,A -85,B 0,C 180,E1 -20610,E2 -20610} C_VEL
LIN {X 0,Y 211.565,Z 469.478,A -85,B 0,C 180,E1 -20611.904,E2 -20611.904} C_VEL
LIN {X 0,Y 211.499,Z 467.755,A -85,B 0,C 180,E1 -20614.431,E2 -20614.431} C_VEL
LIN {X 0,Y 211.722,Z 464.431,A -85,B 0,C 180,E1 -20617.63,E2 -20617.63} C_VEL
LIN {X 0,Y 212.198,Z 460.3,A -85,B 0,C 180,E1 -20620.495,E2 -20620.495} C_VEL
LIN {X 0,Y 213.256,Z 453.932,A -85,B 0,C 180,E1 -20623.823,E2 -20623.823} C_VEL
LIN {X 0,Y 214.745,Z 446.984,A -85,B 0,C 180,E1 -20626.64,E2 -20626.64} C_VEL
LIN {X 0,Y 216.551,Z 438.623,A -85,B 0,C 180,E1 -20629.321,E2 -20629.321} C_VEL
LIN {X 0,Y 218.527,Z 429.281,A -85,B 0,C 180,E1 -20631.706,E2 -20631.706} C_VEL
LIN {X 0,Y 220.507,Z 419.419,A -85,B 0,C 180,E1 -20633.727,E2 -20633.727} C_VEL
LIN {X 0,Y 222.584,Z 408.621,A -85,B 0,C 180,E1 -20635.48,E2 -20635.48} C_VEL
LIN {X 0,Y 224.617,Z 396.55,A -85,B 0,C 180,E1 -20636.98,E2 -20636.98} C_VEL
LIN {X 0,Y 226.15,Z 385.332,A -85,B 0,C 180,E1 -20638.036,E2 -20638.036} C_VEL
LIN {X 0,Y 227.53,Z 372.132,A -85,B 0,C 180,E1 -20638.92,E2 -20638.92} C_VEL
LIN {X 0,Y 228.378,Z 357.792,A -85,B 0,C 180,E1 -20639.496,E2 -20639.496} C_VEL
LIN {X 0,Y 230.171,Z 313.149,A -85,B 0,C 180,E1 -20640.957,E2 -20640.957} C_VEL
LIN {X 0,Y 226.564,Z 285.286,A -85,B 0,C 180,E1 -20642.444,E2 -20642.444} C_VEL
LIN {X 0,Y 218.652,Z 264.612,A -85,B 0,C 180,E1 -20644.303,E2 -20644.303} C_VEL
LIN {X 0,Y 216.179,Z 258.346,A -85,B 0,C 180,E1 -20644.963,E2 -20644.963} C_VEL
LIN {X 0,Y 214.427,Z 250.543,A -85,B 0,C 180,E1 -20648.515,E2 -20648.515} C_VEL
LIN {X 0,Y 213.753,Z 247.862,A -85,B 0,C 180,E1 -20649.876,E2 -20649.876} C_VEL
LIN {X 0,Y 213.698,Z 247.87,A -85,B 0,C 180,E1 -20653.679,E2 -20653.679} C_VEL
LIN {X 0,Y 213.697,Z 247.868,A -85,B 0,C 180,E1 -20656.345,E2 -20656.345} C_VEL
LIN {X 0,Y 213.711,Z 247.864,A -85,B 0,C 180,E1 -20659.143,E2 -20659.143} C_VEL
LIN {X 0,Y 213.754,Z 247.858,A -85,B 0,C 180,E1 -20663.703,E2 -20663.703} C_VEL
LIN {X 0,Y 213.78,Z 247.853,A -85,B 0,C 180,E1 -20668.73,E2 -20668.73} C_VEL
LIN {X 0,Y 213.777,Z 247.853,A -85,B 0,C 180,E1 -20672.586,E2 -20672.586} C_VEL
LIN {X 0,Y 213.804,Z 247.852,A -85,B 0,C 180,E1 -20676.981,E2 -20676.981} C_VEL
LIN {X 0,Y 213.888,Z 247.816,A -85,B 0,C 180,E1 -20682.789,E2 -20682.789} C_VEL
LIN {X 0,Y 213.925,Z 247.833,A -85,B 0,C 180,E1 -20686.695,E2 -20686.695} C_VEL
LIN {X 0,Y 214.124,Z 247.809,A -85,B 0,C 180,E1 -20690.544,E2 -20690.544} C_VEL
LIN {X 0,Y 214.06,Z 247.798,A -85,B 0,C 180,E1 -20694.337,E2 -20694.337} C_VEL
LIN {X 0,Y 214.369,Z 247.75,A -85,B 0,C 180,E1 -20698.111,E2 -20698.111} C_VEL
LIN {X 0,Y 214.502,Z 247.749,A -85,B 0,C 180,E1 -20699.989,E2 -20699.989} C_VEL
LIN {X 0,Y 214.397,Z 247.773,A -85,B 0,C 180,E1 -20701.868,E2 -20701.868} C_VEL
LIN {X 0,Y 214.167,Z 247.802,A -85,B 0,C 180,E1 -20707.531,E2 -20707.531} C_VEL
LIN {X 0,Y 213.98,Z 247.825,A -85,B 0,C 180,E1 -20711.354,E2 -20711.354} C_VEL
LIN {X 0,Y 213.898,Z 247.841,A -85,B 0,C 180,E1 -20715.227,E2 -20715.227} C_VEL
LIN {X 0,Y 213.813,Z 247.84,A -85,B 0,C 180,E1 -20719.177,E2 -20719.177} C_VEL
LIN {X 0,Y 213.781,Z 247.855,A -85,B 0,C 180,E1 -20723.221,E2 -20723.221} C_VEL
LIN {X 0,Y 213.786,Z 247.839,A -85,B 0,C 180,E1 -20727.43,E2 -20727.43} C_VEL
LIN {X 0,Y 213.73,Z 247.822,A -85,B 0,C 180,E1 -20731.729,E2 -20731.729} C_VEL
LIN {X 0,Y 213.709,Z 247.856,A -85,B 0,C 180,E1 -20736.279,E2 -20736.279} C_VEL
LIN {X 0,Y 213.671,Z 247.869,A -85,B 0,C 180,E1 -20741.118,E2 -20741.118} C_VEL
LIN {X 0,Y 213.668,Z 247.863,A -85,B 0,C 180,E1 -20743.67,E2 -20743.67} C_VEL
LIN {X 0,Y 213.667,Z 247.868,A -85,B 0,C 180,E1 -20746.336,E2 -20746.336} C_VEL
LIN {X 0,Y 213.677,Z 247.865,A -85,B 0,C 180,E1 -20749.135,E2 -20749.135} C_VEL
LIN {X 0,Y 213.701,Z 247.866,A -85,B 0,C 180,E1 -20753.704,E2 -20753.704} C_VEL
LIN {X 0,Y 213.736,Z 247.862,A -85,B 0,C 180,E1 -20758.725,E2 -20758.725} C_VEL
LIN {X 0,Y 213.78,Z 247.853,A -85,B 0,C 180,E1 -20762.598,E2 -20762.598} C_VEL
LIN {X 0,Y 213.822,Z 247.853,A -85,B 0,C 180,E1 -20766.937,E2 -20766.937} C_VEL
LIN {X 0,Y 213.92,Z 247.838,A -85,B 0,C 180,E1 -20772.802,E2 -20772.802} C_VEL
LIN {X 0,Y 213.971,Z 247.833,A -85,B 0,C 180,E1 -20778.634,E2 -20778.634} C_VEL
LIN {X 0,Y 214.175,Z 247.804,A -85,B 0,C 180,E1 -20782.458,E2 -20782.458} C_VEL
LIN {X 0,Y 214.398,Z 247.834,A -85,B 0,C 180,E1 -20788.063,E2 -20788.063} C_VEL
LIN {X 0,Y 215.618,Z 250.902,A -85,B 0,C 180,E1 -20788.367,E2 -20788.367} C_VEL
LIN {X 0,Y 221.698,Z 263.247,A -85,B 0,C 180,E1 -20789.711,E2 -20789.711} C_VEL
LIN {X 0,Y 228.761,Z 281.043,A -85,B 0,C 180,E1 -20791.315,E2 -20791.315} C_VEL
LIN {X 0,Y 231.08,Z 287.99,A -85,B 0,C 180,E1 -20791.857,E2 -20791.857} C_VEL
LIN {X 0,Y 228.209,Z 352.061,A -85,B 0,C 180,E1 -20793.973,E2 -20793.973} C_VEL
LIN {X 0,Y 227.081,Z 365.604,A -85,B 0,C 180,E1 -20794.771,E2 -20794.771} C_VEL
LIN {X 0,Y 225.821,Z 377.602,A -85,B 0,C 180,E1 -20795.818,E2 -20795.818} C_VEL
LIN {X 0,Y 224.12,Z 389.449,A -85,B 0,C 180,E1 -20797.205,E2 -20797.205} C_VEL
LIN {X 0,Y 222.224,Z 400.456,A -85,B 0,C 180,E1 -20798.869,E2 -20798.869} C_VEL
LIN {X 0,Y 220.347,Z 410.143,A -85,B 0,C 180,E1 -20800.701,E2 -20800.701} C_VEL
LIN {X 0,Y 218.167,Z 420.064,A -85,B 0,C 180,E1 -20803.032,E2 -20803.032} C_VEL
LIN {X 0,Y 216.386,Z 428.499,A -85,B 0,C 180,E1 -20805.542,E2 -20805.542} C_VEL
LIN {X 0,Y 214.667,Z 436.055,A -85,B 0,C 180,E1 -20808.343,E2 -20808.343} C_VEL
LIN {X 0,Y 213.414,Z 442.213,A -85,B 0,C 180,E1 -20811.237,E2 -20811.237} C_VEL
LIN {X 0,Y 212.418,Z 447.403,A -85,B 0,C 180,E1 -20814.429,E2 -20814.429} C_VEL
LIN {X 0,Y 211.748,Z 451.25,A -85,B 0,C 180,E1 -20817.688,E2 -20817.688} C_VEL
LIN {X 0,Y 211.308,Z 453.33,A -85,B 0,C 180,E1 -20820.173,E2 -20820.173} C_VEL
LIN {X 0,Y 211.161,Z 455.018,A -85,B 0,C 180,E1 -20823.713,E2 -20823.713} C_VEL
LIN {X 0,Y 211.493,Z 455.358,A -85,B 0,C 180,E1 -20827.128,E2 -20827.128} C_VEL
LIN {X 0,Y 212.25,Z 454.479,A -85,B 0,C 180,E1 -20830.417,E2 -20830.417} C_VEL
LIN {X 0,Y 213.468,Z 452.356,A -85,B 0,C 180,E1 -20833.738,E2 -20833.738} C_VEL
LIN {X 0,Y 215.392,Z 448.331,A -85,B 0,C 180,E1 -20837.472,E2 -20837.472} C_VEL
LIN {X 0,Y 217.785,Z 443.189,A -85,B 0,C 180,E1 -20840.757,E2 -20840.757} C_VEL
LIN {X 0,Y 220.374,Z 437.128,A -85,B 0,C 180,E1 -20843.632,E2 -20843.632} C_VEL
LIN {X 0,Y 223.552,Z 429.494,A -85,B 0,C 180,E1 -20846.415,E2 -20846.415} C_VEL
LIN {X 0,Y 226.673,Z 421.262,A -85,B 0,C 180,E1 -20848.779,E2 -20848.779} C_VEL
LIN {X 0,Y 229.623,Z 412.546,A -85,B 0,C 180,E1 -20850.786,E2 -20850.786} C_VEL
LIN {X 0,Y 232.902,Z 401.668,A -85,B 0,C 180,E1 -20852.756,E2 -20852.756} C_VEL
LIN {X 0,Y 235.783,Z 390.282,A -85,B 0,C 180,E1 -20854.374,E2 -20854.374} C_VEL
LIN {X 0,Y 238.252,Z 378.673,A -85,B 0,C 180,E1 -20855.62,E2 -20855.62} C_VEL
LIN {X 0,Y 240.266,Z 365.622,A -85,B 0,C 180,E1 -20856.661,E2 -20856.661} C_VEL
LIN {X 0,Y 241.745,Z 352.172,A -85,B 0,C 180,E1 -20857.37,E2 -20857.37} C_VEL
LIN {X 0,Y 244.99,Z 298.979,A -85,B 0,C 180,E1 -20859.053,E2 -20859.053} C_VEL
LIN {X 0,Y 240.378,Z 288.643,A -85,B 0,C 180,E1 -20860.605,E2 -20860.605} C_VEL
LIN {X 0,Y 235.166,Z 278.692,A -85,B 0,C 180,E1 -20862.429,E2 -20862.429} C_VEL
LIN {X 0,Y 230.786,Z 271.41,A -85,B 0,C 180,E1 -20864.048,E2 -20864.048} C_VEL
LIN {X 0,Y 224.684,Z 262.712,A -85,B 0,C 180,E1 -20866.472,E2 -20866.472} C_VEL
LIN {X 0,Y 222.052,Z 259.09,A -85,B 0,C 180,E1 -20867.617,E2 -20867.617} C_VEL
LIN {X 0,Y 220.747,Z 257.62,A -85,B 0,C 180,E1 -20868.193,E2 -20868.193} C_VEL
LIN {X 0,Y 218.6,Z 254.714,A -85,B 0,C 180,E1 -20869.21,E2 -20869.21} C_VEL
LIN {X 0,Y 217.866,Z 253.236,A -85,B 0,C 180,E1 -20869.603,E2 -20869.603} C_VEL
LIN {X 0,Y 215.59,Z 251.304,A -85,B 0,C 180,E1 -20870.69,E2 -20870.69} C_VEL
LIN {X 0,Y 214.379,Z 248.888,A -85,B 0,C 180,E1 -20871.409,E2 -20871.409} C_VEL
LIN {X 0,Y 214.156,Z 247.801,A -85,B 0,C 180,E1 -20871.638,E2 -20871.638} C_VEL
LIN {X 0,Y 214.434,Z 247.764,A -85,B 0,C 180,E1 -20878.133,E2 -20878.133} C_VEL
LIN {X 0,Y 214.533,Z 247.762,A -85,B 0,C 180,E1 -20880.011,E2 -20880.011} C_VEL
LIN {X 0,Y 214.402,Z 247.766,A -85,B 0,C 180,E1 -20881.889,E2 -20881.889} C_VEL
LIN {X 0,Y 214.187,Z 247.801,A -85,B 0,C 180,E1 -20887.552,E2 -20887.552} C_VEL
LIN {X 0,Y 213.993,Z 247.823,A -85,B 0,C 180,E1 -20891.375,E2 -20891.375} C_VEL
LIN {X 0,Y 213.886,Z 247.834,A -85,B 0,C 180,E1 -20895.25,E2 -20895.25} C_VEL
LIN {X 0,Y 213.797,Z 247.843,A -85,B 0,C 180,E1 -20899.201,E2 -20899.201} C_VEL
LIN {X 0,Y 213.793,Z 247.843,A -85,B 0,C 180,E1 -20903.243,E2 -20903.243} C_VEL
LIN {X 0,Y 213.777,Z 247.848,A -85,B 0,C 180,E1 -20907.426,E2 -20907.426} C_VEL
LIN {X 0,Y 213.767,Z 247.857,A -85,B 0,C 180,E1 -20911.748,E2 -20911.748} C_VEL
LIN {X 0,Y 213.76,Z 247.85,A -85,B 0,C 180,E1 -20914.052,E2 -20914.052} C_VEL
LIN {X 0,Y 213.144,Z 248.28,A -85,B 0,C 180,E1 -20915.128,E2 -20915.128} C_VEL
LIN {X 0,Y 211.27,Z 249.857,A -85,B 0,C 180,E1 -20916.47,E2 -20916.47} C_VEL
LIN {X 0,Y 209.229,Z 252.916,A -85,B 0,C 180,E1 -20918.058,E2 -20918.058} C_VEL
LIN {X 0,Y 209.177,Z 255.123,A -85,B 0,C 180,E1 -20918.979,E2 -20918.979} C_VEL
LIN {X 0,Y 209.504,Z 255.877,A -85,B 0,C 180,E1 -20919.269,E2 -20919.269} C_VEL
LIN {X 0,Y 213.573,Z 261.436,A -85,B 0,C 180,E1 -20921.64,E2 -20921.64} C_VEL
LIN {X 0,Y 217.843,Z 267.734,A -85,B 0,C 180,E1 -20923.839,E2 -20923.839} C_VEL
LIN {X 0,Y 221.667,Z 273.94,A -85,B 0,C 180,E1 -20925.647,E2 -20925.647} C_VEL
LIN {X 0,Y 224.786,Z 279.181,A -85,B 0,C 180,E1 -20927.008,E2 -20927.008} C_VEL
LIN {X 0,Y 229.73,Z 288.287,A -85,B 0,C 180,E1 -20929.035,E2 -20929.035} C_VEL
LIN {X 0,Y 234.978,Z 299.768,A -85,B 0,C 180,E1 -20931.056,E2 -20931.056} C_VEL
LIN {X 0,Y 237.725,Z 307.012,A -85,B 0,C 180,E1 -20932.104,E2 -20932.104} C_VEL
LIN {X 0,Y 238.795,Z 318.047,A -85,B 0,C 180,E1 -20932.888,E2 -20932.888} C_VEL
LIN {X 0,Y 235.711,Z 366.365,A -85,B 0,C 180,E1 -20934.472,E2 -20934.472} C_VEL
LIN {X 0,Y 233.946,Z 379.874,A -85,B 0,C 180,E1 -20935.196,E2 -20935.196} C_VEL
LIN {X 0,Y 231.651,Z 391.877,A -85,B 0,C 180,E1 -20936.12,E2 -20936.12} C_VEL
LIN {X 0,Y 228.692,Z 404.332,A -85,B 0,C 180,E1 -20937.467,E2 -20937.467} C_VEL
LIN {X 0,Y 225.458,Z 415.515,A -85,B 0,C 180,E1 -20939.048,E2 -20939.048} C_VEL
LIN {X 0,Y 222.079,Z 425.683,A -85,B 0,C 180,E1 -20940.886,E2 -20940.886} C_VEL
LIN {X 0,Y 218.463,Z 435.678,A -85,B 0,C 180,E1 -20943.233,E2 -20943.233} C_VEL
LIN {X 0,Y 214.879,Z 444.531,A -85,B 0,C 180,E1 -20945.869,E2 -20945.869} C_VEL
LIN {X 0,Y 211.996,Z 451.703,A -85,B 0,C 180,E1 -20948.614,E2 -20948.614} C_VEL
LIN {X 0,Y 209.5,Z 457.47,A -85,B 0,C 180,E1 -20951.417,E2 -20951.417} C_VEL
LIN {X 0,Y 207.369,Z 462.051,A -85,B 0,C 180,E1 -20954.269,E2 -20954.269} C_VEL
LIN {X 0,Y 205.934,Z 465.567,A -85,B 0,C 180,E1 -20957.184,E2 -20957.184} C_VEL
LIN {X 0,Y 204.994,Z 468.1,A -85,B 0,C 180,E1 -20960.13,E2 -20960.13} C_VEL
LIN {X 0,Y 204.417,Z 470.028,A -85,B 0,C 180,E1 -20964.08,E2 -20964.08} C_VEL
LIN {X 0,Y 204.363,Z 470.408,A -85,B 0,C 180,E1 -20966.056,E2 -20966.056} C_VEL
LIN {X 0,Y 204.418,Z 470.4,A -85,B 0,C 180,E1 -20968.03,E2 -20968.03} C_VEL
LIN {X 0,Y 204.556,Z 469.97,A -85,B 0,C 180,E1 -20970,E2 -20970} C_VEL
LIN {X 0,Y 204.463,Z 469.095,A -85,B 0,C 180,E1 -20971.97,E2 -20971.97} C_VEL
LIN {X 0,Y 204.406,Z 467.574,A -85,B 0,C 180,E1 -20974.265,E2 -20974.265} C_VEL
LIN {X 0,Y 204.554,Z 465.049,A -85,B 0,C 180,E1 -20976.907,E2 -20976.907} C_VEL
LIN {X 0,Y 204.976,Z 461.218,A -85,B 0,C 180,E1 -20979.871,E2 -20979.871} C_VEL
LIN {X 0,Y 205.738,Z 456.215,A -85,B 0,C 180,E1 -20982.829,E2 -20982.829} C_VEL
LIN {X 0,Y 207.079,Z 449.906,A -85,B 0,C 180,E1 -20985.754,E2 -20985.754} C_VEL
LIN {X 0,Y 208.915,Z 441.989,A -85,B 0,C 180,E1 -20988.637,E2 -20988.637} C_VEL
LIN {X 0,Y 210.664,Z 433.765,A -85,B 0,C 180,E1 -20991.043,E2 -20991.043} C_VEL
LIN {X 0,Y 212.822,Z 423.956,A -85,B 0,C 180,E1 -20993.345,E2 -20993.345} C_VEL
LIN {X 0,Y 214.77,Z 414.241,A -85,B 0,C 180,E1 -20995.176,E2 -20995.176} C_VEL
LIN {X 0,Y 216.732,Z 403.821,A -85,B 0,C 180,E1 -20996.738,E2 -20996.738} C_VEL
LIN {X 0,Y 218.658,Z 392.52,A -85,B 0,C 180,E1 -20998.038,E2 -20998.038} C_VEL
LIN {X 0,Y 220.28,Z 379.149,A -85,B 0,C 180,E1 -20999.179,E2 -20999.179} C_VEL
LIN {X 0,Y 221.485,Z 365.886,A -85,B 0,C 180,E1 -20999.918,E2 -20999.918} C_VEL
LIN {X 0,Y 223.714,Z 313.851,A -85,B 0,C 180,E1 -21001.691,E2 -21001.691} C_VEL
LIN {X 0,Y 220.398,Z 287.65,A -85,B 0,C 180,E1 -21003.142,E2 -21003.142} C_VEL
LIN {X 0,Y 212.93,Z 267.932,A -85,B 0,C 180,E1 -21004.971,E2 -21004.971} C_VEL
LIN {X 0,Y 208.958,Z 258.119,A -85,B 0,C 180,E1 -21006.013,E2 -21006.013} C_VEL
LIN {X 0,Y 206.684,Z 248.746,A -85,B 0,C 180,E1 -21010.574,E2 -21010.574} C_VEL
LIN {X 0,Y 206.629,Z 248.749,A -85,B 0,C 180,E1 -21015.582,E2 -21015.582} C_VEL
LIN {X 0,Y 206.657,Z 248.744,A -85,B 0,C 180,E1 -21019.736,E2 -21019.736} C_VEL
LIN {X 0,Y 206.715,Z 248.735,A -85,B 0,C 180,E1 -21024.681,E2 -21024.681} C_VEL
LIN {X 0,Y 206.7,Z 248.736,A -85,B 0,C 180,E1 -21029.324,E2 -21029.324} C_VEL
LIN {X 0,Y 206.682,Z 248.736,A -85,B 0,C 180,E1 -21033.755,E2 -21033.755} C_VEL
LIN {X 0,Y 206.721,Z 248.73,A -85,B 0,C 180,E1 -21038.029,E2 -21038.029} C_VEL
LIN {X 0,Y 206.81,Z 248.695,A -85,B 0,C 180,E1 -21042.18,E2 -21042.18} C_VEL
LIN {X 0,Y 206.866,Z 248.712,A -85,B 0,C 180,E1 -21046.232,E2 -21046.232} C_VEL
LIN {X 0,Y 207.073,Z 248.688,A -85,B 0,C 180,E1 -21050.219,E2 -21050.219} C_VEL
LIN {X 0,Y 207.024,Z 248.673,A -85,B 0,C 180,E1 -21054.144,E2 -21054.144} C_VEL
LIN {X 0,Y 207.311,Z 248.626,A -85,B 0,C 180,E1 -21058.046,E2 -21058.046} C_VEL
LIN {X 0,Y 207.469,Z 248.624,A -85,B 0,C 180,E1 -21059.989,E2 -21059.989} C_VEL
LIN {X 0,Y 207.337,Z 248.653,A -85,B 0,C 180,E1 -21061.931,E2 -21061.931} C_VEL
LIN {X 0,Y 207.113,Z 248.679,A -85,B 0,C 180,E1 -21067.789,E2 -21067.789} C_VEL
LIN {X 0,Y 206.903,Z 248.709,A -85,B 0,C 180,E1 -21071.748,E2 -21071.748} C_VEL
LIN {X 0,Y 206.835,Z 248.717,A -85,B 0,C 180,E1 -21075.761,E2 -21075.761} C_VEL
LIN {X 0,Y 206.74,Z 248.726,A -85,B 0,C 180,E1 -21079.86,E2 -21079.86} C_VEL
LIN {X 0,Y 206.719,Z 248.732,A -85,B 0,C 180,E1 -21084.064,E2 -21084.064} C_VEL
LIN {X 0,Y 206.702,Z 248.717,A -85,B 0,C 180,E1 -21088.411,E2 -21088.411} C_VEL
LIN {X 0,Y 206.665,Z 248.707,A -85,B 0,C 180,E1 -21092.948,E2 -21092.948} C_VEL
LIN {X 0,Y 206.636,Z 248.744,A -85,B 0,C 180,E1 -21097.733,E2 -21097.733} C_VEL
LIN {X 0,Y 206.602,Z 248.746,A -85,B 0,C 180,E1 -21101.552,E2 -21101.552} C_VEL
LIN {X 0,Y 206.595,Z 248.75,A -85,B 0,C 180,E1 -21105.573,E2 -21105.573} C_VEL
LIN {X 0,Y 206.621,Z 248.74,A -85,B 0,C 180,E1 -21109.74,E2 -21109.74} C_VEL
LIN {X 0,Y 206.657,Z 248.744,A -85,B 0,C 180,E1 -21114.681,E2 -21114.681} C_VEL
LIN {X 0,Y 206.67,Z 248.746,A -85,B 0,C 180,E1 -21119.331,E2 -21119.331} C_VEL
LIN {X 0,Y 206.691,Z 248.742,A -85,B 0,C 180,E1 -21123.767,E2 -21123.767} C_VEL
LIN {X 0,Y 206.742,Z 248.733,A -85,B 0,C 180,E1 -21128.042,E2 -21128.042} C_VEL
LIN {X 0,Y 206.835,Z 248.719,A -85,B 0,C 180,E1 -21132.194,E2 -21132.194} C_VEL
LIN {X 0,Y 206.844,Z 248.716,A -85,B 0,C 180,E1 -21136.241,E2 -21136.241} C_VEL
LIN {X 0,Y 207.054,Z 248.691,A -85,B 0,C 180,E1 -21140.229,E2 -21140.229} C_VEL
LIN {X 0,Y 207.024,Z 248.695,A -85,B 0,C 180,E1 -21144.155,E2 -21144.155} C_VEL
LIN {X 0,Y 207.161,Z 248.676,A -85,B 0,C 180,E1 -21146.98,E2 -21146.98} C_VEL
LIN {X 0,Y 208.256,Z 251.592,A -85,B 0,C 180,E1 -21147.298,E2 -21147.298} C_VEL
LIN {X 0,Y 210.696,Z 255.721,A -85,B 0,C 180,E1 -21147.847,E2 -21147.847} C_VEL
LIN {X 0,Y 216.835,Z 268.714,A -85,B 0,C 180,E1 -21149.269,E2 -21149.269} C_VEL
LIN {X 0,Y 223.108,Z 284.845,A -85,B 0,C 180,E1 -21150.75,E2 -21150.75} C_VEL
LIN {X 0,Y 224.592,Z 289.471,A -85,B 0,C 180,E1 -21151.119,E2 -21151.119} C_VEL
LIN {X 0,Y 221.712,Z 352.334,A -85,B 0,C 180,E1 -21153.257,E2 -21153.257} C_VEL
LIN {X 0,Y 220.575,Z 365.571,A -85,B 0,C 180,E1 -21154.054,E2 -21154.054} C_VEL
LIN {X 0,Y 219.18,Z 378.193,A -85,B 0,C 180,E1 -21155.182,E2 -21155.182} C_VEL
LIN {X 0,Y 217.29,Z 390.836,A -85,B 0,C 180,E1 -21156.733,E2 -21156.733} C_VEL
LIN {X 0,Y 215.339,Z 401.644,A -85,B 0,C 180,E1 -21158.445,E2 -21158.445} C_VEL
LIN {X 0,Y 213.18,Z 412.187,A -85,B 0,C 180,E1 -21160.556,E2 -21160.556} C_VEL
LIN {X 0,Y 210.946,Z 421.834,A -85,B 0,C 180,E1 -21162.996,E2 -21162.996} C_VEL
LIN {X 0,Y 209.14,Z 430.032,A -85,B 0,C 180,E1 -21165.594,E2 -21165.594} C_VEL
LIN {X 0,Y 207.456,Z 437.375,A -85,B 0,C 180,E1 -21168.503,E2 -21168.503} C_VEL
LIN {X 0,Y 206.391,Z 442.31,A -85,B 0,C 180,E1 -21170.949,E2 -21170.949} C_VEL
LIN {X 0,Y 205.353,Z 447.552,A -85,B 0,C 180,E1 -21174.247,E2 -21174.247} C_VEL
LIN {X 0,Y 204.826,Z 450.73,A -85,B 0,C 180,E1 -21176.892,E2 -21176.892} C_VEL
LIN {X 0,Y 204.161,Z 453.815,A -85,B 0,C 180,E1 -21180.644,E2 -21180.644} C_VEL
LIN {X 0,Y 204.082,Z 455.379,A -85,B 0,C 180,E1 -21184.285,E2 -21184.285} C_VEL
LIN {X 0,Y 204.589,Z 455.558,A -85,B 0,C 180,E1 -21188.193,E2 -21188.193} C_VEL
LIN {X 0,Y 205.383,Z 454.632,A -85,B 0,C 180,E1 -21191.186,E2 -21191.186} C_VEL
LIN {X 0,Y 206.641,Z 452.535,A -85,B 0,C 180,E1 -21194.44,E2 -21194.44} C_VEL
LIN {X 0,Y 208.495,Z 448.999,A -85,B 0,C 180,E1 -21197.864,E2 -21197.864} C_VEL
LIN {X 0,Y 210.481,Z 445.01,A -85,B 0,C 180,E1 -21200.64,E2 -21200.64} C_VEL
LIN {X 0,Y 213.04,Z 439.458,A -85,B 0,C 180,E1 -21203.589,E2 -21203.589} C_VEL
LIN {X 0,Y 216.315,Z 432.323,A -85,B 0,C 180,E1 -21206.488,E2 -21206.488} C_VEL
LIN {X 0,Y 219.314,Z 425.051,A -85,B 0,C 180,E1 -21208.823,E2 -21208.823} C_VEL
LIN {X 0,Y 222.693,Z 415.993,A -85,B 0,C 180,E1 -21211.133,E2 -21211.133} C_VEL
LIN {X 0,Y 226.253,Z 405.195,A -85,B 0,C 180,E1 -21213.29,E2 -21213.29} C_VEL
LIN {X 0,Y 229.18,Z 394.926,A -85,B 0,C 180,E1 -21214.896,E2 -21214.896} C_VEL
LIN {X 0,Y 231.808,Z 383.787,A -85,B 0,C 180,E1 -21216.255,E2 -21216.255} C_VEL
LIN {X 0,Y 234.239,Z 370.457,A -85,B 0,C 180,E1 -21217.472,E2 -21217.472} C_VEL
LIN {X 0,Y 235.956,Z 357.732,A -85,B 0,C 180,E1 -21218.267,E2 -21218.267} C_VEL
LIN {X 0,Y 237.2,Z 341.978,A -85,B 0,C 180,E1 -21218.859,E2 -21218.859} C_VEL
LIN {X 0,Y 239.789,Z 301.301,A -85,B 0,C 180,E1 -21220.148,E2 -21220.148} C_VEL
LIN {X 0,Y 234.356,Z 289.393,A -85,B 0,C 180,E1 -21222.11,E2 -21222.11} C_VEL
LIN {X 0,Y 228.713,Z 279.07,A -85,B 0,C 180,E1 -21224.257,E2 -21224.257} C_VEL
LIN {X 0,Y 223.481,Z 271.239,A -85,B 0,C 180,E1 -21226.374,E2 -21226.374} C_VEL
LIN {X 0,Y 221.285,Z 268.134,A -85,B 0,C 180,E1 -21227.334,E2 -21227.334} C_VEL
LIN {X 0,Y 218.395,Z 264.038,A -85,B 0,C 180,E1 -21228.675,E2 -21228.675} C_VEL
LIN {X 0,Y 215.824,Z 260.777,A -85,B 0,C 180,E1 -21229.923,E2 -21229.923} C_VEL
LIN {X 0,Y 214.815,Z 259.227,A -85,B 0,C 180,E1 -21230.46,E2 -21230.46} C_VEL
LIN {X 0,Y 212.409,Z 256.454,A -85,B 0,C 180,E1 -21231.748,E2 -21231.748} C_VEL
LIN {X 0,Y 211.229,Z 254.261,A -85,B 0,C 180,E1 -21232.483,E2 -21232.483} C_VEL
LIN {X 0,Y 208.695,Z 252.433,A -85,B 0,C 180,E1 -21233.91,E2 -21233.91} C_VEL
LIN {X 0,Y 207.329,Z 250.043,A -85,B 0,C 180,E1 -21234.845,E2 -21234.845} C_VEL
LIN {X 0,Y 207.044,Z 248.686,A -85,B 0,C 180,E1 -21235.143,E2 -21235.143} C_VEL
LIN {X 0,Y 207.37,Z 248.644,A -85,B 0,C 180,E1 -21238.069,E2 -21238.069} C_VEL
LIN {X 0,Y 207.498,Z 248.638,A -85,B 0,C 180,E1 -21240.011,E2 -21240.011} C_VEL
LIN {X 0,Y 207.044,Z 248.694,A -85,B 0,C 180,E1 -21243.904,E2 -21243.904} C_VEL
LIN {X 0,Y 207.131,Z 248.683,A -85,B 0,C 180,E1 -21247.811,E2 -21247.811} C_VEL
LIN {X 0,Y 206.914,Z 248.708,A -85,B 0,C 180,E1 -21251.769,E2 -21251.769} C_VEL
LIN {X 0,Y 206.818,Z 248.719,A -85,B 0,C 180,E1 -21255.785,E2 -21255.785} C_VEL
LIN {X 0,Y 206.719,Z 248.73,A -85,B 0,C 180,E1 -21259.886,E2 -21259.886} C_VEL
LIN {X 0,Y 206.706,Z 248.733,A -85,B 0,C 180,E1 -21264.09,E2 -21264.09} C_VEL
LIN {X 0,Y 206.683,Z 248.739,A -85,B 0,C 180,E1 -21268.439,E2 -21268.439} C_VEL
LIN {X 0,Y 206.692,Z 248.741,A -85,B 0,C 180,E1 -21273.333,E2 -21273.333} C_VEL
LIN {X 0,Y 208.588,Z 254.256,A -85,B 0,C 180,E1 -21278.663,E2 -21278.663} C_VEL
LIN {X 0,Y 209.504,Z 255.877,A -85,B 0,C 180,E1 -21279.269,E2 -21279.269} C_VEL
LIN {X 0,Y 211.267,Z 259.592,A -85,B 0,C 180,E1 -21280.431,E2 -21280.431} C_VEL
LIN {X 0,Y 213.747,Z 266.926,A -85,B 0,C 180,E1 -21282.101,E2 -21282.101} C_VEL
LIN {X 0,Y 215.721,Z 273.096,A -85,B 0,C 180,E1 -21283.352,E2 -21283.352} C_VEL
LIN {X 0,Y 218.136,Z 278.837,A -85,B 0,C 180,E1 -21284.667,E2 -21284.667} C_VEL
LIN {X 0,Y 221.691,Z 285.086,A -85,B 0,C 180,E1 -21286.327,E2 -21286.327} C_VEL
LIN {X 0,Y 226.523,Z 294.369,A -85,B 0,C 180,E1 -21288.404,E2 -21288.404} C_VEL
LIN {X 0,Y 231.569,Z 306.16,A -85,B 0,C 180,E1 -21290.474,E2 -21290.474} C_VEL
LIN {X 0,Y 232.956,Z 310.133,A -85,B 0,C 180,E1 -21291.042,E2 -21291.042} C_VEL
LIN {X 0,Y 233.718,Z 319.841,A -85,B 0,C 180,E1 -21291.718,E2 -21291.718} C_VEL
LIN {X 0,Y 230.561,Z 366.252,A -85,B 0,C 180,E1 -21293.271,E2 -21293.271} C_VEL
LIN {X 0,Y 228.637,Z 380.252,A -85,B 0,C 180,E1 -21294.042,E2 -21294.042} C_VEL
LIN {X 0,Y 226.307,Z 391.676,A -85,B 0,C 180,E1 -21294.935,E2 -21294.935} C_VEL
LIN {X 0,Y 223.246,Z 404.072,A -85,B 0,C 180,E1 -21296.301,E2 -21296.301} C_VEL
LIN {X 0,Y 219.869,Z 415.255,A -85,B 0,C 180,E1 -21297.9,E2 -21297.9} C_VEL
LIN {X 0,Y 216.362,Z 425.419,A -85,B 0,C 180,E1 -21299.771,E2 -21299.771} C_VEL
LIN {X 0,Y 212.832,Z 434.608,A -85,B 0,C 180,E1 -21301.931,E2 -21301.931} C_VEL
LIN {X 0,Y 208.993,Z 443.595,A -85,B 0,C 180,E1 -21304.612,E2 -21304.612} C_VEL
LIN {X 0,Y 206.063,Z 450.524,A -85,B 0,C 180,E1 -21307.277,E2 -21307.277} C_VEL
LIN {X 0,Y 203.546,Z 455.828,A -85,B 0,C 180,E1 -21309.802,E2 -21309.802} C_VEL
LIN {X 0,Y 201.222,Z 460.687,A -85,B 0,C 180,E1 -21312.731,E2 -21312.731} C_VEL
LIN {X 0,Y 199.39,Z 464.463,A -85,B 0,C 180,E1 -21315.716,E2 -21315.716} C_VEL
LIN {X 0,Y 198.598,Z 466.436,A -85,B 0,C 180,E1 -21317.742,E2 -21317.742} C_VEL
LIN {X 0,Y 197.977,Z 467.981,A -85,B 0,C 180,E1 -21319.777,E2 -21319.777} C_VEL
LIN {X 0,Y 197.332,Z 469.817,A -85,B 0,C 180,E1 -21323.867,E2 -21323.867} C_VEL
LIN {X 0,Y 197.274,Z 470.179,A -85,B 0,C 180,E1 -21326.078,E2 -21326.078} C_VEL
LIN {X 0,Y 197.321,Z 470.107,A -85,B 0,C 180,E1 -21327.959,E2 -21327.959} C_VEL
LIN {X 0,Y 197.472,Z 469.617,A -85,B 0,C 180,E1 -21330,E2 -21330} C_VEL
LIN {X 0,Y 197.364,Z 468.708,A -85,B 0,C 180,E1 -21332.041,E2 -21332.041} C_VEL
LIN {X 0,Y 197.339,Z 467.317,A -85,B 0,C 180,E1 -21334.188,E2 -21334.188} C_VEL
LIN {X 0,Y 197.485,Z 464.555,A -85,B 0,C 180,E1 -21337.155,E2 -21337.155} C_VEL
LIN {X 0,Y 197.948,Z 460.647,A -85,B 0,C 180,E1 -21340.225,E2 -21340.225} C_VEL
LIN {X 0,Y 198.956,Z 454.584,A -85,B 0,C 180,E1 -21343.794,E2 -21343.794} C_VEL
LIN {X 0,Y 200.516,Z 447.902,A -85,B 0,C 180,E1 -21346.807,E2 -21346.807} C_VEL
LIN {X 0,Y 202.465,Z 439.568,A -85,B 0,C 180,E1 -21349.782,E2 -21349.782} C_VEL
LIN {X 0,Y 204.409,Z 431.011,A -85,B 0,C 180,E1 -21352.222,E2 -21352.222} C_VEL
LIN {X 0,Y 206.507,Z 421.613,A -85,B 0,C 180,E1 -21354.371,E2 -21354.371} C_VEL
LIN {X 0,Y 208.369,Z 412.839,A -85,B 0,C 180,E1 -21356.006,E2 -21356.006} C_VEL
LIN {X 0,Y 210.406,Z 402.072,A -85,B 0,C 180,E1 -21357.61,E2 -21357.61} C_VEL
LIN {X 0,Y 212.543,Z 389.217,A -85,B 0,C 180,E1 -21359.055,E2 -21359.055} C_VEL
LIN {X 0,Y 213.974,Z 377.036,A -85,B 0,C 180,E1 -21360.058,E2 -21360.058} C_VEL
LIN {X 0,Y 215.154,Z 363.635,A -85,B 0,C 180,E1 -21360.757,E2 -21360.757} C_VEL
LIN {X 0,Y 217.296,Z 314.7,A -85,B 0,C 180,E1 -21362.464,E2 -21362.464} C_VEL
LIN {X 0,Y 214.226,Z 289.912,A -85,B 0,C 180,E1 -21363.875,E2 -21363.875} C_VEL
LIN {X 0,Y 207.02,Z 270.833,A -85,B 0,C 180,E1 -21365.718,E2 -21365.718} C_VEL
LIN {X 0,Y 201.612,Z 257.812,A -85,B 0,C 180,E1 -21367.194,E2 -21367.194} C_VEL
LIN {X 0,Y 199.609,Z 249.621,A -85,B 0,C 180,E1 -21371.369,E2 -21371.369} C_VEL
LIN {X 0,Y 199.575,Z 249.628,A -85,B 0,C 180,E1 -21375.215,E2 -21375.215} C_VEL
LIN {X 0,Y 199.575,Z 249.625,A -85,B 0,C 180,E1 -21377.991,E2 -21377.991} C_VEL
LIN {X 0,Y 199.611,Z 249.62,A -85,B 0,C 180,E1 -21380.766,E2 -21380.766} C_VEL
LIN {X 0,Y 199.623,Z 249.623,A -85,B 0,C 180,E1 -21385.704,E2 -21385.704} C_VEL
LIN {X 0,Y 199.695,Z 249.608,A -85,B 0,C 180,E1 -21388.125,E2 -21388.125} C_VEL
LIN {X 0,Y 199.632,Z 249.615,A -85,B 0,C 180,E1 -21392.753,E2 -21392.753} C_VEL
LIN {X 0,Y 199.679,Z 249.612,A -85,B 0,C 180,E1 -21397.211,E2 -21397.211} C_VEL
LIN {X 0,Y 199.752,Z 249.573,A -85,B 0,C 180,E1 -21401.793,E2 -21401.793} C_VEL
LIN {X 0,Y 199.804,Z 249.587,A -85,B 0,C 180,E1 -21405.735,E2 -21405.735} C_VEL
LIN {X 0,Y 200.025,Z 249.567,A -85,B 0,C 180,E1 -21409.871,E2 -21409.871} C_VEL
LIN {X 0,Y 199.989,Z 249.549,A -85,B 0,C 180,E1 -21413.937,E2 -21413.937} C_VEL
LIN {X 0,Y 200.255,Z 249.502,A -85,B 0,C 180,E1 -21417.978,E2 -21417.978} C_VEL
LIN {X 0,Y 200.436,Z 249.498,A -85,B 0,C 180,E1 -21419.989,E2 -21419.989} C_VEL
LIN {X 0,Y 199.98,Z 249.574,A -85,B 0,C 180,E1 -21424.019,E2 -21424.019} C_VEL
LIN {X 0,Y 200.061,Z 249.556,A -85,B 0,C 180,E1 -21428.066,E2 -21428.066} C_VEL
LIN {X 0,Y 199.853,Z 249.587,A -85,B 0,C 180,E1 -21432.168,E2 -21432.168} C_VEL
LIN {X 0,Y 199.777,Z 249.594,A -85,B 0,C 180,E1 -21436.333,E2 -21436.333} C_VEL
LIN {X 0,Y 199.659,Z 249.608,A -85,B 0,C 180,E1 -21440.596,E2 -21440.596} C_VEL
LIN {X 0,Y 199.635,Z 249.615,A -85,B 0,C 180,E1 -21444.975,E2 -21444.975} C_VEL
LIN {X 0,Y 199.601,Z 249.588,A -85,B 0,C 180,E1 -21449.519,E2 -21449.519} C_VEL
LIN {X 0,Y 199.636,Z 249.575,A -85,B 0,C 180,E1 -21452.341,E2 -21452.341} C_VEL
LIN {X 0,Y 199.586,Z 249.615,A -85,B 0,C 180,E1 -21456.754,E2 -21456.754} C_VEL
LIN {X 0,Y 199.563,Z 249.628,A -85,B 0,C 180,E1 -21459.321,E2 -21459.321} C_VEL
LIN {X 0,Y 199.535,Z 249.624,A -85,B 0,C 180,E1 -21462.299,E2 -21462.299} C_VEL
LIN {X 0,Y 199.542,Z 249.626,A -85,B 0,C 180,E1 -21465.219,E2 -21465.219} C_VEL
LIN {X 0,Y 199.54,Z 249.628,A -85,B 0,C 180,E1 -21467.996,E2 -21467.996} C_VEL
LIN {X 0,Y 199.569,Z 249.618,A -85,B 0,C 180,E1 -21470.76,E2 -21470.76} C_VEL
LIN {X 0,Y 199.569,Z 249.622,A -85,B 0,C 180,E1 -21475.706,E2 -21475.706} C_VEL
LIN {X 0,Y 199.649,Z 249.616,A -85,B 0,C 180,E1 -21478.129,E2 -21478.129} C_VEL
LIN {X 0,Y 199.643,Z 249.615,A -85,B 0,C 180,E1 -21482.766,E2 -21482.766} C_VEL
LIN {X 0,Y 199.71,Z 249.609,A -85,B 0,C 180,E1 -21487.226,E2 -21487.226} C_VEL
LIN {X 0,Y 199.79,Z 249.597,A -85,B 0,C 180,E1 -21491.717,E2 -21491.717} C_VEL
LIN {X 0,Y 199.787,Z 249.596,A -85,B 0,C 180,E1 -21495.745,E2 -21495.745} C_VEL
LIN {X 0,Y 200.021,Z 249.567,A -85,B 0,C 180,E1 -21499.882,E2 -21499.882} C_VEL
LIN {X 0,Y 199.986,Z 249.569,A -85,B 0,C 180,E1 -21503.948,E2 -21503.948} C_VEL
LIN {X 0,Y 199.993,Z 249.573,A -85,B 0,C 180,E1 -21505.844,E2 -21505.844} C_VEL
LIN {X 0,Y 201.186,Z 252.649,A -85,B 0,C 180,E1 -21506.207,E2 -21506.207} C_VEL
LIN {X 0,Y 205.777,Z 260.716,A -85,B 0,C 180,E1 -21507.307,E2 -21507.307} C_VEL
LIN {X 0,Y 211.066,Z 271.948,A -85,B 0,C 180,E1 -21508.588,E2 -21508.588} C_VEL
LIN {X 0,Y 217.129,Z 287.68,A -85,B 0,C 180,E1 -21510.078,E2 -21510.078} C_VEL
LIN {X 0,Y 218.292,Z 291.333,A -85,B 0,C 180,E1 -21510.378,E2 -21510.378} C_VEL
LIN {X 0,Y 215.247,Z 352.782,A -85,B 0,C 180,E1 -21512.514,E2 -21512.514} C_VEL
LIN {X 0,Y 214.086,Z 365.486,A -85,B 0,C 180,E1 -21513.293,E2 -21513.293} C_VEL
LIN {X 0,Y 212.687,Z 377.871,A -85,B 0,C 180,E1 -21514.418,E2 -21514.418} C_VEL
LIN {X 0,Y 211.037,Z 388.751,A -85,B 0,C 180,E1 -21515.734,E2 -21515.734} C_VEL
LIN {X 0,Y 208.985,Z 399.978,A -85,B 0,C 180,E1 -21517.487,E2 -21517.487} C_VEL
LIN {X 0,Y 206.704,Z 411.005,A -85,B 0,C 180,E1 -21519.682,E2 -21519.682} C_VEL
LIN {X 0,Y 204.578,Z 419.923,A -85,B 0,C 180,E1 -21521.895,E2 -21521.895} C_VEL
LIN {X 0,Y 202.675,Z 428.334,A -85,B 0,C 180,E1 -21524.508,E2 -21524.508} C_VEL
LIN {X 0,Y 200.923,Z 435.559,A -85,B 0,C 180,E1 -21527.296,E2 -21527.296} C_VEL
LIN {X 0,Y 199.383,Z 442.377,A -85,B 0,C 180,E1 -21530.639,E2 -21530.639} C_VEL
LIN {X 0,Y 198.311,Z 447.678,A -85,B 0,C 180,E1 -21534.052,E2 -21534.052} C_VEL
LIN {X 0,Y 197.556,Z 451.6,A -85,B 0,C 180,E1 -21537.546,E2 -21537.546} C_VEL
LIN {X 0,Y 197.024,Z 454.285,A -85,B 0,C 180,E1 -21541.147,E2 -21541.147} C_VEL
LIN {X 0,Y 197.041,Z 455.736,A -85,B 0,C 180,E1 -21544.905,E2 -21544.905} C_VEL
LIN {X 0,Y 197.568,Z 455.848,A -85,B 0,C 180,E1 -21548.524,E2 -21548.524} C_VEL
LIN {X 0,Y 198.624,Z 454.629,A -85,B 0,C 180,E1 -21552.242,E2 -21552.242} C_VEL
LIN {X 0,Y 199.953,Z 452.567,A -85,B 0,C 180,E1 -21555.354,E2 -21555.354} C_VEL
LIN {X 0,Y 201.776,Z 449.31,A -85,B 0,C 180,E1 -21558.582,E2 -21558.582} C_VEL
LIN {X 0,Y 204.585,Z 444.114,A -85,B 0,C 180,E1 -21562.193,E2 -21562.193} C_VEL
LIN {X 0,Y 207.506,Z 438.228,A -85,B 0,C 180,E1 -21565.213,E2 -21565.213} C_VEL
LIN {X 0,Y 210.727,Z 431.321,A -85,B 0,C 180,E1 -21567.941,E2 -21567.941} C_VEL
LIN {X 0,Y 214.322,Z 422.898,A -85,B 0,C 180,E1 -21570.55,E2 -21570.55} C_VEL
LIN {X 0,Y 217.955,Z 413.359,A -85,B 0,C 180,E1 -21572.878,E2 -21572.878} C_VEL
LIN {X 0,Y 221.361,Z 403.214,A -85,B 0,C 180,E1 -21574.799,E2 -21574.799} C_VEL
LIN {X 0,Y 224.664,Z 391.497,A -85,B 0,C 180,E1 -21576.544,E2 -21576.544} C_VEL
LIN {X 0,Y 227.525,Z 379.211,A -85,B 0,C 180,E1 -21577.917,E2 -21577.917} C_VEL
LIN {X 0,Y 229.684,Z 366.688,A -85,B 0,C 180,E1 -21578.945,E2 -21578.945} C_VEL
LIN {X 0,Y 231.288,Z 353.597,A -85,B 0,C 180,E1 -21579.671,E2 -21579.671} C_VEL
LIN {X 0,Y 234.635,Z 303.651,A -85,B 0,C 180,E1 -21581.326,E2 -21581.326} C_VEL
LIN {X 0,Y 229.825,Z 293.063,A -85,B 0,C 180,E1 -21583.173,E2 -21583.173} C_VEL
LIN {X 0,Y 224.572,Z 283.388,A -85,B 0,C 180,E1 -21585.309,E2 -21585.309} C_VEL
LIN {X 0,Y 218.85,Z 274.547,A -85,B 0,C 180,E1 -21587.827,E2 -21587.827} C_VEL
LIN {X 0,Y 215.004,Z 269.374,A -85,B 0,C 180,E1 -21589.67,E2 -21589.67} C_VEL
LIN {X 0,Y 212.013,Z 265.179,A -85,B 0,C 180,E1 -21591.275,E2 -21591.275} C_VEL
LIN {X 0,Y 209.504,Z 261.873,A -85,B 0,C 180,E1 -21592.724,E2 -21592.724} C_VEL
LIN {X 0,Y 208.882,Z 260.738,A -85,B 0,C 180,E1 -21593.127,E2 -21593.127} C_VEL
LIN {X 0,Y 206.264,Z 258.452,A -85,B 0,C 180,E1 -21594.696,E2 -21594.696} C_VEL
LIN {X 0,Y 204.723,Z 255.637,A -85,B 0,C 180,E1 -21595.828,E2 -21595.828} C_VEL
LIN {X 0,Y 201.901,Z 253.209,A -85,B 0,C 180,E1 -21597.892,E2 -21597.892} C_VEL
LIN {X 0,Y 200.69,Z 250.934,A -85,B 0,C 180,E1 -21599.008,E2 -21599.008} C_VEL
LIN {X 0,Y 200.399,Z 249.516,A -85,B 0,C 180,E1 -21599.446,E2 -21599.446} C_VEL
LIN {X 0,Y 200.284,Z 249.524,A -85,B 0,C 180,E1 -21602.022,E2 -21602.022} C_VEL
LIN {X 0,Y 200.078,Z 249.562,A -85,B 0,C 180,E1 -21608.088,E2 -21608.088} C_VEL
LIN {X 0,Y 199.863,Z 249.59,A -85,B 0,C 180,E1 -21612.191,E2 -21612.191} C_VEL
LIN {X 0,Y 199.754,Z 249.604,A -85,B 0,C 180,E1 -21616.359,E2 -21616.359} C_VEL
LIN {X 0,Y 199.651,Z 249.616,A -85,B 0,C 180,E1 -21620.621,E2 -21620.621} C_VEL
LIN {X 0,Y 199.628,Z 249.614,A -85,B 0,C 180,E1 -21625.001,E2 -21625.001} C_VEL
LIN {X 0,Y 199.616,Z 249.66,A -85,B 0,C 180,E1 -21629.196,E2 -21629.196} C_VEL
LIN {X 0,Y 200.974,Z 253.358,A -85,B 0,C 180,E1 -21633.95,E2 -21633.95} C_VEL
LIN {X 0,Y 204.534,Z 258.65,A -85,B 0,C 180,E1 -21636.822,E2 -21636.822} C_VEL
LIN {X 0,Y 206.403,Z 260.802,A -85,B 0,C 180,E1 -21638.057,E2 -21638.057} C_VEL
LIN {X 0,Y 209.886,Z 265.925,A -85,B 0,C 180,E1 -21640.266,E2 -21640.266} C_VEL
LIN {X 0,Y 212.222,Z 269.523,A -85,B 0,C 180,E1 -21641.628,E2 -21641.628} C_VEL
LIN {X 0,Y 214.926,Z 273.592,A -85,B 0,C 180,E1 -21643.069,E2 -21643.069} C_VEL
LIN {X 0,Y 218.136,Z 278.837,A -85,B 0,C 180,E1 -21644.667,E2 -21644.667} C_VEL
LIN {X 0,Y 219.198,Z 281.939,A -85,B 0,C 180,E1 -21645.256,E2 -21645.256} C_VEL
LIN {X 0,Y 220.014,Z 288.104,A -85,B 0,C 180,E1 -21645.93,E2 -21645.93} C_VEL
LIN {X 0,Y 220.84,Z 294.328,A -85,B 0,C 180,E1 -21646.586,E2 -21646.586} C_VEL
LIN {X 0,Y 221.947,Z 297.522,A -85,B 0,C 180,E1 -21647.138,E2 -21647.138} C_VEL
LIN {X 0,Y 226.863,Z 309.112,A -85,B 0,C 180,E1 -21649.31,E2 -21649.31} C_VEL
LIN {X 0,Y 228.182,Z 312.674,A -85,B 0,C 180,E1 -21649.882,E2 -21649.882} C_VEL
LIN {X 0,Y 228.816,Z 320.439,A -85,B 0,C 180,E1 -21650.458,E2 -21650.458} C_VEL
LIN {X 0,Y 225.623,Z 365.548,A -85,B 0,C 180,E1 -21651.98,E2 -21651.98} C_VEL
LIN {X 0,Y 223.618,Z 379.67,A -85,B 0,C 180,E1 -21652.754,E2 -21652.754} C_VEL
LIN {X 0,Y 221.089,Z 391.667,A -85,B 0,C 180,E1 -21653.698,E2 -21653.698} C_VEL
LIN {X 0,Y 217.896,Z 403.991,A -85,B 0,C 180,E1 -21655.076,E2 -21655.076} C_VEL
LIN {X 0,Y 214.362,Z 415.104,A -85,B 0,C 180,E1 -21656.692,E2 -21656.692} C_VEL
LIN {X 0,Y 210.724,Z 425.203,A -85,B 0,C 180,E1 -21658.594,E2 -21658.594} C_VEL
LIN {X 0,Y 206.612,Z 435.164,A -85,B 0,C 180,E1 -21661.007,E2 -21661.007} C_VEL
LIN {X 0,Y 202.618,Z 444.016,A -85,B 0,C 180,E1 -21663.754,E2 -21663.754} C_VEL
LIN {X 0,Y 199.368,Z 451.187,A -85,B 0,C 180,E1 -21666.651,E2 -21666.651} C_VEL
LIN {X 0,Y 196.876,Z 456.026,A -85,B 0,C 180,E1 -21669.086,E2 -21669.086} C_VEL
LIN {X 0,Y 194.437,Z 460.784,A -85,B 0,C 180,E1 -21672.108,E2 -21672.108} C_VEL
LIN {X 0,Y 192.488,Z 464.457,A -85,B 0,C 180,E1 -21675.193,E2 -21675.193} C_VEL
LIN {X 0,Y 191.64,Z 466.377,A -85,B 0,C 180,E1 -21677.289,E2 -21677.289} C_VEL
LIN {X 0,Y 190.498,Z 468.918,A -85,B 0,C 180,E1 -21681.514,E2 -21681.514} C_VEL
LIN {X 0,Y 190.19,Z 469.913,A -85,B 0,C 180,E1 -21685.762,E2 -21685.762} C_VEL
LIN {X 0,Y 190.227,Z 469.789,A -85,B 0,C 180,E1 -21687.883,E2 -21687.883} C_VEL
LIN {X 0,Y 190.39,Z 469.258,A -85,B 0,C 180,E1 -21690,E2 -21690} C_VEL
LIN {X 0,Y 190.263,Z 467.07,A -85,B 0,C 180,E1 -21694.067,E2 -21694.067} C_VEL
LIN {X 0,Y 190.44,Z 464.037,A -85,B 0,C 180,E1 -21697.421,E2 -21697.421} C_VEL
LIN {X 0,Y 190.94,Z 460.041,A -85,B 0,C 180,E1 -21700.605,E2 -21700.605} C_VEL
LIN {X 0,Y 192.026,Z 453.833,A -85,B 0,C 180,E1 -21704.302,E2 -21704.302} C_VEL
LIN {X 0,Y 193.673,Z 447.042,A -85,B 0,C 180,E1 -21707.42,E2 -21707.42} C_VEL
LIN {X 0,Y 195.681,Z 438.565,A -85,B 0,C 180,E1 -21710.498,E2 -21710.498} C_VEL
LIN {X 0,Y 197.783,Z 429.81,A -85,B 0,C 180,E1 -21713.008,E2 -21713.008} C_VEL
LIN {X 0,Y 200.229,Z 419.023,A -85,B 0,C 180,E1 -21715.465,E2 -21715.465} C_VEL
LIN {X 0,Y 202.519,Z 408.33,A -85,B 0,C 180,E1 -21717.374,E2 -21717.374} C_VEL
LIN {X 0,Y 204.748,Z 396.413,A -85,B 0,C 180,E1 -21719.001,E2 -21719.001} C_VEL
LIN {X 0,Y 206.602,Z 384.115,A -85,B 0,C 180,E1 -21720.256,E2 -21720.256} C_VEL
LIN {X 0,Y 208.047,Z 371.692,A -85,B 0,C 180,E1 -21721.149,E2 -21721.149} C_VEL
LIN {X 0,Y 208.953,Z 357.615,A -85,B 0,C 180,E1 -21721.774,E2 -21721.774} C_VEL
LIN {X 0,Y 210.892,Z 315.433,A -85,B 0,C 180,E1 -21723.27,E2 -21723.27} C_VEL
LIN {X 0,Y 208.014,Z 291.933,A -85,B 0,C 180,E1 -21724.66,E2 -21724.66} C_VEL
LIN {X 0,Y 200.346,Z 271.693,A -85,B 0,C 180,E1 -21726.727,E2 -21726.727} C_VEL
LIN {X 0,Y 195.24,Z 260.057,A -85,B 0,C 180,E1 -21728.113,E2 -21728.113} C_VEL
LIN {X 0,Y 194.301,Z 257.623,A -85,B 0,C 180,E1 -21728.402,E2 -21728.402} C_VEL
LIN {X 0,Y 192.539,Z 250.499,A -85,B 0,C 180,E1 -21732.227,E2 -21732.227} C_VEL
LIN {X 0,Y 192.487,Z 250.511,A -85,B 0,C 180,E1 -21736.904,E2 -21736.904} C_VEL
LIN {X 0,Y 192.556,Z 250.501,A -85,B 0,C 180,E1 -21741.637,E2 -21741.637} C_VEL
LIN {X 0,Y 192.607,Z 250.495,A -85,B 0,C 180,E1 -21746.804,E2 -21746.804} C_VEL
LIN {X 0,Y 192.619,Z 250.492,A -85,B 0,C 180,E1 -21751.673,E2 -21751.673} C_VEL
LIN {X 0,Y 192.666,Z 250.485,A -85,B 0,C 180,E1 -21756.332,E2 -21756.332} C_VEL
LIN {X 0,Y 192.702,Z 250.45,A -85,B 0,C 180,E1 -21761.481,E2 -21761.481} C_VEL
LIN {X 0,Y 192.73,Z 250.464,A -85,B 0,C 180,E1 -21765.2,E2 -21765.2} C_VEL
LIN {X 0,Y 192.948,Z 250.45,A -85,B 0,C 180,E1 -21769.556,E2 -21769.556} C_VEL
LIN {X 0,Y 192.954,Z 250.426,A -85,B 0,C 180,E1 -21773.715,E2 -21773.715} C_VEL
LIN {X 0,Y 193.202,Z 250.378,A -85,B 0,C 180,E1 -21777.904,E2 -21777.904} C_VEL
LIN {X 0,Y 193.402,Z 250.373,A -85,B 0,C 180,E1 -21779.988,E2 -21779.988} C_VEL
LIN {X 0,Y 192.928,Z 250.452,A -85,B 0,C 180,E1 -21784.166,E2 -21784.166} C_VEL
LIN {X 0,Y 193.012,Z 250.433,A -85,B 0,C 180,E1 -21788.362,E2 -21788.362} C_VEL
LIN {X 0,Y 192.78,Z 250.468,A -85,B 0,C 180,E1 -21792.622,E2 -21792.622} C_VEL
LIN {X 0,Y 192.734,Z 250.471,A -85,B 0,C 180,E1 -21796.947,E2 -21796.947} C_VEL
LIN {X 0,Y 192.592,Z 250.491,A -85,B 0,C 180,E1 -21801.388,E2 -21801.388} C_VEL
LIN {X 0,Y 192.62,Z 250.488,A -85,B 0,C 180,E1 -21804.197,E2 -21804.197} C_VEL
LIN {X 0,Y 192.602,Z 250.463,A -85,B 0,C 180,E1 -21808.868,E2 -21808.868} C_VEL
LIN {X 0,Y 192.566,Z 250.46,A -85,B 0,C 180,E1 -21813.176,E2 -21813.176} C_VEL
LIN {X 0,Y 192.51,Z 250.502,A -85,B 0,C 180,E1 -21818.344,E2 -21818.344} C_VEL
LIN {X 0,Y 192.453,Z 250.504,A -85,B 0,C 180,E1 -21823.085,E2 -21823.085} C_VEL
LIN {X 0,Y 192.453,Z 250.512,A -85,B 0,C 180,E1 -21826.896,E2 -21826.896} C_VEL
LIN {X 0,Y 192.51,Z 250.502,A -85,B 0,C 180,E1 -21831.639,E2 -21831.639} C_VEL
LIN {X 0,Y 192.554,Z 250.495,A -85,B 0,C 180,E1 -21836.806,E2 -21836.806} C_VEL
LIN {X 0,Y 192.62,Z 250.49,A -85,B 0,C 180,E1 -21841.685,E2 -21841.685} C_VEL
LIN {X 0,Y 192.669,Z 250.489,A -85,B 0,C 180,E1 -21846.344,E2 -21846.344} C_VEL
LIN {X 0,Y 192.735,Z 250.478,A -85,B 0,C 180,E1 -21851.409,E2 -21851.409} C_VEL
LIN {X 0,Y 192.717,Z 250.48,A -85,B 0,C 180,E1 -21855.21,E2 -21855.21} C_VEL
LIN {X 0,Y 192.932,Z 250.45,A -85,B 0,C 180,E1 -21859.506,E2 -21859.506} C_VEL
LIN {X 0,Y 193.011,Z 250.442,A -85,B 0,C 180,E1 -21861.625,E2 -21861.625} C_VEL
LIN {X 0,Y 192.957,Z 250.449,A -85,B 0,C 180,E1 -21864.646,E2 -21864.646} C_VEL
LIN {X 0,Y 194.028,Z 253.415,A -85,B 0,C 180,E1 -21865.028,E2 -21865.028} C_VEL
LIN {X 0,Y 200.96,Z 265.71,A -85,B 0,C 180,E1 -21866.761,E2 -21866.761} C_VEL
LIN {X 0,Y 205.639,Z 276.091,A -85,B 0,C 180,E1 -21867.956,E2 -21867.956} C_VEL
LIN {X 0,Y 211.156,Z 290.423,A -85,B 0,C 180,E1 -21869.376,E2 -21869.376} C_VEL
LIN {X 0,Y 211.889,Z 292.849,A -85,B 0,C 180,E1 -21869.58,E2 -21869.58} C_VEL
LIN {X 0,Y 208.826,Z 352.479,A -85,B 0,C 180,E1 -21871.701,E2 -21871.701} C_VEL
LIN {X 0,Y 207.637,Z 365.178,A -85,B 0,C 180,E1 -21872.485,E2 -21872.485} C_VEL
LIN {X 0,Y 206.167,Z 377.913,A -85,B 0,C 180,E1 -21873.664,E2 -21873.664} C_VEL
LIN {X 0,Y 204.275,Z 389.835,A -85,B 0,C 180,E1 -21875.159,E2 -21875.159} C_VEL
LIN {X 0,Y 202.119,Z 401.047,A -85,B 0,C 180,E1 -21876.99,E2 -21876.99} C_VEL
LIN {X 0,Y 200.07,Z 410.608,A -85,B 0,C 180,E1 -21878.954,E2 -21878.954} C_VEL
LIN {X 0,Y 197.831,Z 419.754,A -85,B 0,C 180,E1 -21881.267,E2 -21881.267} C_VEL
LIN {X 0,Y 195.681,Z 428.896,A -85,B 0,C 180,E1 -21884.196,E2 -21884.196} C_VEL
LIN {X 0,Y 193.735,Z 436.628,A -85,B 0,C 180,E1 -21887.334,E2 -21887.334} C_VEL
LIN {X 0,Y 192.387,Z 442.422,A -85,B 0,C 180,E1 -21890.306,E2 -21890.306} C_VEL
LIN {X 0,Y 191.258,Z 447.784,A -85,B 0,C 180,E1 -21893.841,E2 -21893.841} C_VEL
LIN {X 0,Y 190.41,Z 451.945,A -85,B 0,C 180,E1 -21897.678,E2 -21897.678} C_VEL
LIN {X 0,Y 189.883,Z 454.751,A -85,B 0,C 180,E1 -21901.677,E2 -21901.677} C_VEL
LIN {X 0,Y 190.015,Z 456.073,A -85,B 0,C 180,E1 -21905.566,E2 -21905.566} C_VEL
LIN {X 0,Y 190.62,Z 456.058,A -85,B 0,C 180,E1 -21909.286,E2 -21909.286} C_VEL
LIN {X 0,Y 191.727,Z 454.885,A -85,B 0,C 180,E1 -21912.872,E2 -21912.872} C_VEL
LIN {X 0,Y 193.45,Z 452.397,A -85,B 0,C 180,E1 -21916.6,E2 -21916.6} C_VEL
LIN {X 0,Y 196.034,Z 448.104,A -85,B 0,C 180,E1 -21920.612,E2 -21920.612} C_VEL
LIN {X 0,Y 199.155,Z 442.418,A -85,B 0,C 180,E1 -21924.255,E2 -21924.255} C_VEL
LIN {X 0,Y 202.54,Z 436.04,A -85,B 0,C 180,E1 -21927.292,E2 -21927.292} C_VEL
LIN {X 0,Y 206.423,Z 427.921,A -85,B 0,C 180,E1 -21930.246,E2 -21930.246} C_VEL
LIN {X 0,Y 210.113,Z 419.338,A -85,B 0,C 180,E1 -21932.693,E2 -21932.693} C_VEL
LIN {X 0,Y 213.517,Z 410.56,A -85,B 0,C 180,E1 -21934.679,E2 -21934.679} C_VEL
LIN {X 0,Y 217.05,Z 399.998,A -85,B 0,C 180,E1 -21936.585,E2 -21936.585} C_VEL
LIN {X 0,Y 220.374,Z 387.952,A -85,B 0,C 180,E1 -21938.249,E2 -21938.249} C_VEL
LIN {X 0,Y 223.155,Z 375.469,A -85,B 0,C 180,E1 -21939.539,E2 -21939.539} C_VEL
LIN {X 0,Y 225.26,Z 362.324,A -85,B 0,C 180,E1 -21940.505,E2 -21940.505} C_VEL
LIN {X 0,Y 226.76,Z 348.226,A -85,B 0,C 180,E1 -21941.15,E2 -21941.15} C_VEL
LIN {X 0,Y 229.622,Z 306.111,A -85,B 0,C 180,E1 -21942.54,E2 -21942.54} C_VEL
LIN {X 0,Y 225.176,Z 296.207,A -85,B 0,C 180,E1 -21944.395,E2 -21944.395} C_VEL
LIN {X 0,Y 220.591,Z 287.763,A -85,B 0,C 180,E1 -21946.375,E2 -21946.375} C_VEL
LIN {X 0,Y 215.218,Z 279.558,A -85,B 0,C 180,E1 -21948.896,E2 -21948.896} C_VEL
LIN {X 0,Y 212.15,Z 275.198,A -85,B 0,C 180,E1 -21950.477,E2 -21950.477} C_VEL
LIN {X 0,Y 209.435,Z 271.262,A -85,B 0,C 180,E1 -21952.015,E2 -21952.015} C_VEL
LIN {X 0,Y 206.684,Z 267.324,A -85,B 0,C 180,E1 -21953.713,E2 -21953.713} C_VEL
LIN {X 0,Y 203.837,Z 264.453,A -85,B 0,C 180,E1 -21955.541,E2 -21955.541} C_VEL
LIN {X 0,Y 202.409,Z 261.898,A -85,B 0,C 180,E1 -21956.652,E2 -21956.652} C_VEL
LIN {X 0,Y 200.039,Z 259.725,A -85,B 0,C 180,E1 -21958.502,E2 -21958.502} C_VEL
LIN {X 0,Y 198.495,Z 256.714,A -85,B 0,C 180,E1 -21960.011,E2 -21960.011} C_VEL
LIN {X 0,Y 198.214,Z 256.245,A -85,B 0,C 180,E1 -21960.291,E2 -21960.291} C_VEL
LIN {X 0,Y 194.642,Z 254.224,A -85,B 0,C 180,E1 -21963.893,E2 -21963.893} C_VEL
LIN {X 0,Y 193.292,Z 251.894,A -85,B 0,C 180,E1 -21965.946,E2 -21965.946} C_VEL
LIN {X 0,Y 192.974,Z 250.435,A -85,B 0,C 180,E1 -21966.809,E2 -21966.809} C_VEL
LIN {X 0,Y 192.938,Z 250.438,A -85,B 0,C 180,E1 -21970.505,E2 -21970.505} C_VEL
LIN {X 0,Y 192.731,Z 250.465,A -85,B 0,C 180,E1 -21974.8,E2 -21974.8} C_VEL
LIN {X 0,Y 192.631,Z 250.478,A -85,B 0,C 180,E1 -21979.181,E2 -21979.181} C_VEL
LIN {X 0,Y 192.665,Z 250.625,A -85,B 0,C 180,E1 -21983.099,E2 -21983.099} C_VEL
LIN {X 0,Y 193.081,Z 252.402,A -85,B 0,C 180,E1 -21986.346,E2 -21986.346} C_VEL
LIN {X 0,Y 195.755,Z 256.228,A -85,B 0,C 180,E1 -21990.058,E2 -21990.058} C_VEL
LIN {X 0,Y 199.228,Z 260.175,A -85,B 0,C 180,E1 -21993.432,E2 -21993.432} C_VEL
LIN {X 0,Y 203.151,Z 265.812,A -85,B 0,C 180,E1 -21996.66,E2 -21996.66} C_VEL
LIN {X 0,Y 204.434,Z 267.64,A -85,B 0,C 180,E1 -21997.572,E2 -21997.572} C_VEL
LIN {X 0,Y 208.488,Z 273.678,A -85,B 0,C 180,E1 -22000.199,E2 -22000.199} C_VEL
LIN {X 0,Y 211.973,Z 279.26,A -85,B 0,C 180,E1 -22002.227,E2 -22002.227} C_VEL
LIN {X 0,Y 215.771,Z 285.749,A -85,B 0,C 180,E1 -22004.212,E2 -22004.212} C_VEL
LIN {X 0,Y 219.478,Z 292.56,A -85,B 0,C 180,E1 -22006.015,E2 -22006.015} C_VEL
LIN {X 0,Y 221.947,Z 297.522,A -85,B 0,C 180,E1 -22007.138,E2 -22007.138} C_VEL
LIN {X 0,Y 223.021,Z 300.68,A -85,B 0,C 180,E1 -22007.664,E2 -22007.664} C_VEL
LIN {X 0,Y 223.497,Z 304.362,A -85,B 0,C 180,E1 -22008.023,E2 -22008.023} C_VEL
LIN {X 0,Y 223.799,Z 317.657,A -85,B 0,C 180,E1 -22008.86,E2 -22008.86} C_VEL
LIN {X 0,Y 224.02,Z 321.98,A -85,B 0,C 180,E1 -22009.165,E2 -22009.165} C_VEL
LIN {X 0,Y 220.72,Z 365.666,A -85,B 0,C 180,E1 -22010.667,E2 -22010.667} C_VEL
LIN {X 0,Y 218.696,Z 379.236,A -85,B 0,C 180,E1 -22011.419,E2 -22011.419} C_VEL
LIN {X 0,Y 215.982,Z 391.647,A -85,B 0,C 180,E1 -22012.403,E2 -22012.403} C_VEL
LIN {X 0,Y 212.671,Z 403.916,A -85,B 0,C 180,E1 -22013.794,E2 -22013.794} C_VEL
LIN {X 0,Y 208.952,Z 415.003,A -85,B 0,C 180,E1 -22015.419,E2 -22015.419} C_VEL
LIN {X 0,Y 205.128,Z 425.07,A -85,B 0,C 180,E1 -22017.343,E2 -22017.343} C_VEL
LIN {X 0,Y 201.221,Z 434.191,A -85,B 0,C 180,E1 -22019.574,E2 -22019.574} C_VEL
LIN {X 0,Y 196.949,Z 443.13,A -85,B 0,C 180,E1 -22022.362,E2 -22022.362} C_VEL
LIN {X 0,Y 193.243,Z 450.64,A -85,B 0,C 180,E1 -22025.418,E2 -22025.418} C_VEL
LIN {X 0,Y 190.249,Z 456.223,A -85,B 0,C 180,E1 -22028.322,E2 -22028.322} C_VEL
LIN {X 0,Y 187.685,Z 460.883,A -85,B 0,C 180,E1 -22031.441,E2 -22031.441} C_VEL
LIN {X 0,Y 185.602,Z 464.467,A -85,B 0,C 180,E1 -22034.63,E2 -22034.63} C_VEL
LIN {X 0,Y 184.682,Z 466.308,A -85,B 0,C 180,E1 -22036.802,E2 -22036.802} C_VEL
LIN {X 0,Y 183.453,Z 468.753,A -85,B 0,C 180,E1 -22041.186,E2 -22041.186} C_VEL
LIN {X 0,Y 183.167,Z 469.401,A -85,B 0,C 180,E1 -22043.39,E2 -22043.39} C_VEL
LIN {X 0,Y 183.081,Z 469.602,A -85,B 0,C 180,E1 -22046.591,E2 -22046.591} C_VEL
LIN {X 0,Y 183.309,Z 468.9,A -85,B 0,C 180,E1 -22050,E2 -22050} C_VEL
LIN {X 0,Y 183.174,Z 466.868,A -85,B 0,C 180,E1 -22053.868,E2 -22053.868} C_VEL
LIN {X 0,Y 183.375,Z 463.503,A -85,B 0,C 180,E1 -22057.709,E2 -22057.709} C_VEL
LIN {X 0,Y 183.921,Z 459.414,A -85,B 0,C 180,E1 -22061.015,E2 -22061.015} C_VEL
LIN {X 0,Y 185.121,Z 453.083,A -85,B 0,C 180,E1 -22064.848,E2 -22064.848} C_VEL
LIN {X 0,Y 186.83,Z 446.176,A -85,B 0,C 180,E1 -22068.079,E2 -22068.079} C_VEL
LIN {X 0,Y 188.6,Z 439.225,A -85,B 0,C 180,E1 -22070.687,E2 -22070.687} C_VEL
LIN {X 0,Y 190.765,Z 430.569,A -85,B 0,C 180,E1 -22073.33,E2 -22073.33} C_VEL
LIN {X 0,Y 193.012,Z 421.185,A -85,B 0,C 180,E1 -22075.619,E2 -22075.619} C_VEL
LIN {X 0,Y 195.014,Z 412.43,A -85,B 0,C 180,E1 -22077.354,E2 -22077.354} C_VEL
LIN {X 0,Y 197.491,Z 399.92,A -85,B 0,C 180,E1 -22079.295,E2 -22079.295} C_VEL
LIN {X 0,Y 199.601,Z 387.75,A -85,B 0,C 180,E1 -22080.7,E2 -22080.7} C_VEL
LIN {X 0,Y 201.278,Z 374.233,A -85,B 0,C 180,E1 -22081.801,E2 -22081.801} C_VEL
LIN {X 0,Y 202.389,Z 361.164,A -85,B 0,C 180,E1 -22082.472,E2 -22082.472} C_VEL
LIN {X 0,Y 204.49,Z 315.933,A -85,B 0,C 180,E1 -22084.135,E2 -22084.135} C_VEL
LIN {X 0,Y 201.915,Z 294.286,A -85,B 0,C 180,E1 -22085.466,E2 -22085.466} C_VEL
LIN {X 0,Y 194.545,Z 274.723,A -85,B 0,C 180,E1 -22087.541,E2 -22087.541} C_VEL
LIN {X 0,Y 189.726,Z 263.652,A -85,B 0,C 180,E1 -22088.916,E2 -22088.916} C_VEL
LIN {X 0,Y 186.938,Z 257.259,A -85,B 0,C 180,E1 -22089.792,E2 -22089.792} C_VEL
LIN {X 0,Y 185.458,Z 251.385,A -85,B 0,C 180,E1 -22093.091,E2 -22093.091} C_VEL
LIN {X 0,Y 185.456,Z 251.386,A -85,B 0,C 180,E1 -22096.976,E2 -22096.976} C_VEL
LIN {X 0,Y 185.468,Z 251.383,A -85,B 0,C 180,E1 -22099.882,E2 -22099.882} C_VEL
LIN {X 0,Y 185.517,Z 251.377,A -85,B 0,C 180,E1 -22102.705,E2 -22102.705} C_VEL
LIN {X 0,Y 185.541,Z 251.371,A -85,B 0,C 180,E1 -22107.962,E2 -22107.962} C_VEL
LIN {X 0,Y 185.499,Z 251.374,A -85,B 0,C 180,E1 -22112.946,E2 -22112.946} C_VEL
LIN {X 0,Y 185.554,Z 251.367,A -85,B 0,C 180,E1 -22117.731,E2 -22117.731} C_VEL
LIN {X 0,Y 185.655,Z 251.325,A -85,B 0,C 180,E1 -22122.36,E2 -22122.36} C_VEL
LIN {X 0,Y 185.713,Z 251.347,A -85,B 0,C 180,E1 -22126.864,E2 -22126.864} C_VEL
LIN {X 0,Y 185.969,Z 251.313,A -85,B 0,C 180,E1 -22131.294,E2 -22131.294} C_VEL
LIN {X 0,Y 186.149,Z 251.253,A -85,B 0,C 180,E1 -22137.824,E2 -22137.824} C_VEL
LIN {X 0,Y 186.368,Z 251.247,A -85,B 0,C 180,E1 -22139.988,E2 -22139.988} C_VEL
LIN {X 0,Y 185.876,Z 251.33,A -85,B 0,C 180,E1 -22144.324,E2 -22144.324} C_VEL
LIN {X 0,Y 185.962,Z 251.311,A -85,B 0,C 180,E1 -22148.682,E2 -22148.682} C_VEL
LIN {X 0,Y 185.708,Z 251.351,A -85,B 0,C 180,E1 -22153.111,E2 -22153.111} C_VEL
LIN {X 0,Y 185.669,Z 251.344,A -85,B 0,C 180,E1 -22157.613,E2 -22157.613} C_VEL
LIN {X 0,Y 185.553,Z 251.369,A -85,B 0,C 180,E1 -22162.242,E2 -22162.242} C_VEL
LIN {X 0,Y 185.527,Z 251.359,A -85,B 0,C 180,E1 -22167.022,E2 -22167.022} C_VEL
LIN {X 0,Y 185.505,Z 251.329,A -85,B 0,C 180,E1 -22172.016,E2 -22172.016} C_VEL
LIN {X 0,Y 185.468,Z 251.376,A -85,B 0,C 180,E1 -22177.304,E2 -22177.304} C_VEL
LIN {X 0,Y 185.43,Z 251.386,A -85,B 0,C 180,E1 -22180.712,E2 -22180.712} C_VEL
LIN {X 0,Y 185.422,Z 251.387,A -85,B 0,C 180,E1 -22186.046,E2 -22186.046} C_VEL
LIN {X 0,Y 185.427,Z 251.379,A -85,B 0,C 180,E1 -22189.886,E2 -22189.886} C_VEL
LIN {X 0,Y 185.465,Z 251.382,A -85,B 0,C 180,E1 -22192.704,E2 -22192.704} C_VEL
LIN {X 0,Y 185.5,Z 251.379,A -85,B 0,C 180,E1 -22197.967,E2 -22197.967} C_VEL
LIN {X 0,Y 185.538,Z 251.377,A -85,B 0,C 180,E1 -22200.569,E2 -22200.569} C_VEL
LIN {X 0,Y 185.561,Z 251.377,A -85,B 0,C 180,E1 -22205.379,E2 -22205.379} C_VEL
LIN {X 0,Y 185.664,Z 251.361,A -85,B 0,C 180,E1 -22211.096,E2 -22211.096} C_VEL
LIN {X 0,Y 185.676,Z 251.361,A -85,B 0,C 180,E1 -22214.636,E2 -22214.636} C_VEL
LIN {X 0,Y 185.875,Z 251.329,A -85,B 0,C 180,E1 -22219.357,E2 -22219.357} C_VEL
LIN {X 0,Y 185.906,Z 251.343,A -85,B 0,C 180,E1 -22223.42,E2 -22223.42} C_VEL
LIN {X 0,Y 186.957,Z 254.235,A -85,B 0,C 180,E1 -22223.767,E2 -22223.767} C_VEL
LIN {X 0,Y 195.448,Z 269.432,A -85,B 0,C 180,E1 -22226.027,E2 -22226.027} C_VEL
LIN {X 0,Y 199.821,Z 279.091,A -85,B 0,C 180,E1 -22227.183,E2 -22227.183} C_VEL
LIN {X 0,Y 205.441,Z 293.925,A -85,B 0,C 180,E1 -22228.702,E2 -22228.702} C_VEL
LIN {X 0,Y 202.392,Z 352.829,A -85,B 0,C 180,E1 -22230.87,E2 -22230.87} C_VEL
LIN {X 0,Y 201.15,Z 365.662,A -85,B 0,C 180,E1 -22231.689,E2 -22231.689} C_VEL
LIN {X 0,Y 199.636,Z 378.322,A -85,B 0,C 180,E1 -22232.901,E2 -22232.901} C_VEL
LIN {X 0,Y 197.621,Z 390.486,A -85,B 0,C 180,E1 -22234.481,E2 -22234.481} C_VEL
LIN {X 0,Y 195.289,Z 402.104,A -85,B 0,C 180,E1 -22236.457,E2 -22236.457} C_VEL
LIN {X 0,Y 192.948,Z 412.48,A -85,B 0,C 180,E1 -22238.707,E2 -22238.707} C_VEL
LIN {X 0,Y 190.612,Z 421.506,A -85,B 0,C 180,E1 -22241.161,E2 -22241.161} C_VEL
LIN {X 0,Y 188.437,Z 430.36,A -85,B 0,C 180,E1 -22244.203,E2 -22244.203} C_VEL
LIN {X 0,Y 186.451,Z 438.064,A -85,B 0,C 180,E1 -22247.55,E2 -22247.55} C_VEL
LIN {X 0,Y 184.896,Z 444.439,A -85,B 0,C 180,E1 -22251.167,E2 -22251.167} C_VEL
LIN {X 0,Y 183.95,Z 449.345,A -85,B 0,C 180,E1 -22254.851,E2 -22254.851} C_VEL
LIN {X 0,Y 183.217,Z 452.537,A -85,B 0,C 180,E1 -22258.117,E2 -22258.117} C_VEL
LIN {X 0,Y 182.783,Z 455.21,A -85,B 0,C 180,E1 -22262.26,E2 -22262.26} C_VEL
LIN {X 0,Y 182.996,Z 456.376,A -85,B 0,C 180,E1 -22266.269,E2 -22266.269} C_VEL
LIN {X 0,Y 183.828,Z 456.192,A -85,B 0,C 180,E1 -22270.535,E2 -22270.535} C_VEL
LIN {X 0,Y 184.989,Z 455.019,A -85,B 0,C 180,E1 -22273.815,E2 -22273.815} C_VEL
LIN {X 0,Y 186.705,Z 452.692,A -85,B 0,C 180,E1 -22277.367,E2 -22277.367} C_VEL
LIN {X 0,Y 189.278,Z 448.761,A -85,B 0,C 180,E1 -22281.235,E2 -22281.235} C_VEL
LIN {X 0,Y 192.769,Z 442.852,A -85,B 0,C 180,E1 -22285.192,E2 -22285.192} C_VEL
LIN {X 0,Y 195.999,Z 437.202,A -85,B 0,C 180,E1 -22288.006,E2 -22288.006} C_VEL
LIN {X 0,Y 199.594,Z 430.238,A -85,B 0,C 180,E1 -22290.745,E2 -22290.745} C_VEL
LIN {X 0,Y 203.508,Z 421.857,A -85,B 0,C 180,E1 -22293.338,E2 -22293.338} C_VEL
LIN {X 0,Y 207.417,Z 412.497,A -85,B 0,C 180,E1 -22295.587,E2 -22295.587} C_VEL
LIN {X 0,Y 211.109,Z 402.27,A -85,B 0,C 180,E1 -22297.525,E2 -22297.525} C_VEL
LIN {X 0,Y 214.477,Z 391.104,A -85,B 0,C 180,E1 -22299.191,E2 -22299.191} C_VEL
LIN {X 0,Y 217.547,Z 378.714,A -85,B 0,C 180,E1 -22300.565,E2 -22300.565} C_VEL
LIN {X 0,Y 219.837,Z 366.392,A -85,B 0,C 180,E1 -22301.574,E2 -22301.574} C_VEL
LIN {X 0,Y 221.508,Z 353.669,A -85,B 0,C 180,E1 -22302.276,E2 -22302.276} C_VEL
LIN {X 0,Y 224.802,Z 308.742,A -85,B 0,C 180,E1 -22303.81,E2 -22303.81} C_VEL
LIN {X 0,Y 220.949,Z 300.131,A -85,B 0,C 180,E1 -22305.518,E2 -22305.518} C_VEL
LIN {X 0,Y 217.029,Z 292.768,A -85,B 0,C 180,E1 -22307.348,E2 -22307.348} C_VEL
LIN {X 0,Y 212.218,Z 285.215,A -85,B 0,C 180,E1 -22309.728,E2 -22309.728} C_VEL
LIN {X 0,Y 209.337,Z 280.971,A -85,B 0,C 180,E1 -22311.322,E2 -22311.322} C_VEL
LIN {X 0,Y 206.641,Z 277.028,A -85,B 0,C 180,E1 -22312.93,E2 -22312.93} C_VEL
LIN {X 0,Y 204.057,Z 273.347,A -85,B 0,C 180,E1 -22314.611,E2 -22314.611} C_VEL
LIN {X 0,Y 201.394,Z 270.284,A -85,B 0,C 180,E1 -22316.479,E2 -22316.479} C_VEL
LIN {X 0,Y 200.4,Z 268.438,A -85,B 0,C 180,E1 -22317.31,E2 -22317.31} C_VEL
LIN {X 0,Y 197.929,Z 265.833,A -85,B 0,C 180,E1 -22319.376,E2 -22319.376} C_VEL
LIN {X 0,Y 196.455,Z 263.053,A -85,B 0,C 180,E1 -22320.895,E2 -22320.895} C_VEL
LIN {X 0,Y 193.074,Z 260.826,A -85,B 0,C 180,E1 -22324.579,E2 -22324.579} C_VEL
LIN {X 0,Y 191.753,Z 258.222,A -85,B 0,C 180,E1 -22326.787,E2 -22326.787} C_VEL
LIN {X 0,Y 191.392,Z 257.339,A -85,B 0,C 180,E1 -22327.51,E2 -22327.51} C_VEL
LIN {X 0,Y 188.844,Z 256.414,A -85,B 0,C 180,E1 -22335.112,E2 -22335.112} C_VEL
LIN {X 0,Y 190.033,Z 257.073,A -85,B 0,C 180,E1 -22342.4,E2 -22342.4} C_VEL
LIN {X 0,Y 191.862,Z 259.444,A -85,B 0,C 180,E1 -22346.088,E2 -22346.088} C_VEL
LIN {X 0,Y 194.334,Z 263.088,A -85,B 0,C 180,E1 -22349.656,E2 -22349.656} C_VEL
LIN {X 0,Y 197.373,Z 266.675,A -85,B 0,C 180,E1 -22352.769,E2 -22352.769} C_VEL
LIN {X 0,Y 201.313,Z 272.444,A -85,B 0,C 180,E1 -22356.161,E2 -22356.161} C_VEL
LIN {X 0,Y 205.976,Z 279.761,A -85,B 0,C 180,E1 -22359.434,E2 -22359.434} C_VEL
LIN {X 0,Y 209.127,Z 284.967,A -85,B 0,C 180,E1 -22361.367,E2 -22361.367} C_VEL
LIN {X 0,Y 213.958,Z 293.548,A -85,B 0,C 180,E1 -22364.019,E2 -22364.019} C_VEL
LIN {X 0,Y 218.805,Z 303.582,A -85,B 0,C 180,E1 -22366.448,E2 -22366.448} C_VEL
LIN {X 0,Y 223.291,Z 314.796,A -85,B 0,C 180,E1 -22368.545,E2 -22368.545} C_VEL
LIN {X 0,Y 223.675,Z 316.24,A -85,B 0,C 180,E1 -22368.744,E2 -22368.744} C_VEL
LIN {X 0,Y 223.799,Z 317.657,A -85,B 0,C 180,E1 -22368.86,E2 -22368.86} C_VEL
LIN {X 0,Y 223.849,Z 321.434,A -85,B 0,C 180,E1 -22369.084,E2 -22369.084} C_VEL
LIN {X 0,Y 223.338,Z 325.294,A -85,B 0,C 180,E1 -22369.142,E2 -22369.142} C_VEL
LIN {X 0,Y 221.329,Z 332.95,A -85,B 0,C 180,E1 -22368.957,E2 -22368.957} C_VEL
